KUKA KRL program: EPS_2_251112_SAMH01_A_20250918124112.src

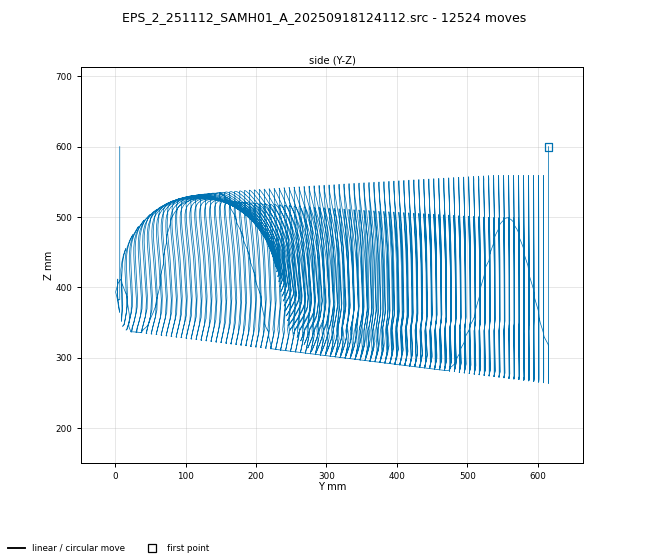
[picture p0: tool path of EPS_2_251112_SAMH01_A_20250918124112.src, 12524 of 12526 moves have a stored position in this frame; points joined in program order, loops and branches not executed]
&ACCESS RVP
&REL 4
&COMMENT QRS 19112012
&PARAM EDITMASK = *
DEF PART()
EXT BAS (BAS_COMMAND :IN,REAL :IN )
INT I
BAS (#INITMOV,0 )

;KUKA QRS Post kuka4.cps  Date:22-06-2017 !

File_ID=2848

QRS_PRE_INIT()

;Init var - Until changes are made in qrs_pre_init
Outlet_Square_prg=0
Inlet_1_Square_prg=0
Inlet_2_Square_prg=0
Inlet_3_Square_prg=0
Inlet_4_Square_prg=0
Inlet_5_Square_prg=0

Outlet_1={X 0.000, Y 535.490, Z 458.500, B 0.000, E1 0.000 }
Inlet_1={X 0.000, Y 540.090, Z 424.000, B 0.000, E1 110.000 }
Outlet_1_type=201
Inlet_1_type=150
;QRS#1=Sidecore dimensions
;QRS#2=200-8" PVC SDR 35
;QRS#3=150-6" PVC SDR 28
;QRS#4=
;QRS#5=
;QRS#6=
;QRS#7=
;QRS#8=
;QRS#9=12-08 PSX
;QRS#10=10-06 PSX
;QRS#11=
;QRS#12=
;QRS#13=
;QRS#14=
;QRS#15=
;QRS#16=1220x127x838 2,75'
;QRS#17=EPS Height
;QRS#18=559
;QRS#19=*
;QRS#20= UPDATED VERSION 22-06-2017
;QRS#21=*
Outlet_Square=0100
Inlet_1_Square=070
Inlet_2_Square=0
Inlet_3_Square=0
Inlet_4_Square=0
Inlet_5_Square=0
Mill_Square=1
Outlet_Square_Prg=204
Inlet_1_Square_prg=203

QRS_INIT()

$ADVANCE=5

; T1
PTP {E1 173.706,E2 173.706}
PTP {X 0,Y 615.438,A -85,B 0,C 180,E1 173.706,E2 173.706,E3 0,E4 0,E5 0,E6 0}
QRS_SPEED_INIT()
LIN {X 0,Y 615.438,Z 600,A -85,B 0,C 180,E1 173.706,E2 173.706,E3 0,E4 0,E5 0,E6 0} C_VEL
LIN {X 0,Y 615.438,Z 326.206,A -85,B 0,C 180,E1 173.706,E2 173.706} C_VEL
LIN {X 0,Y 615.438,Z 317.812,A -85,B 0,C 180,E1 173.706,E2 173.706} C_VEL
LIN {X 0,Y 615.44,Z 316.11,A -85,B 0,C 180,E1 173.422,E2 173.422} C_VEL
LIN {X 0,Y 615.492,Z 334.71,A -85,B 0,C 180,E1 170.635,E2 170.635} C_VEL
LIN {X 0,Y 615.479,Z 338.467,A -85,B 0,C 180,E1 170.075,E2 170.075} C_VEL
LIN {X 0,Y 615.469,Z 414.985,A -85,B 0,C 180,E1 169.169,E2 169.169} C_VEL
LIN {X 0,Y 615.464,Z 424.01,A -85,B 0,C 180,E1 168.989,E2 168.989} C_VEL
LIN {X 0,Y 615.468,Z 433.065,A -85,B 0,C 180,E1 168.723,E2 168.723} C_VEL
LIN {X 0,Y 615.491,Z 441.502,A -85,B 0,C 180,E1 168.389,E2 168.389} C_VEL
LIN {X 0,Y 615.495,Z 449.816,A -85,B 0,C 180,E1 167.972,E2 167.972} C_VEL
LIN {X 0,Y 615.478,Z 457.873,A -85,B 0,C 180,E1 167.469,E2 167.469} C_VEL
LIN {X 0,Y 615.498,Z 466.559,A -85,B 0,C 180,E1 166.799,E2 166.799} C_VEL
LIN {X 0,Y 615.497,Z 474.267,A -85,B 0,C 180,E1 166.046,E2 166.046} C_VEL
LIN {X 0,Y 615.495,Z 480.527,A -85,B 0,C 180,E1 165.282,E2 165.282} C_VEL
LIN {X 0,Y 615.495,Z 484.105,A -85,B 0,C 180,E1 164.774,E2 164.774} C_VEL
LIN {X 0,Y 615.494,Z 489.374,A -85,B 0,C 180,E1 163.824,E2 163.824} C_VEL
LIN {X 0,Y 615.496,Z 492.626,A -85,B 0,C 180,E1 163.072,E2 163.072} C_VEL
LIN {X 0,Y 615.496,Z 495.783,A -85,B 0,C 180,E1 162.043,E2 162.043} C_VEL
LIN {X 0,Y 615.487,Z 497.204,A -85,B 0,C 180,E1 161.354,E2 161.354} C_VEL
LIN {X 0,Y 615.491,Z 498.08,A -85,B 0,C 180,E1 160.662,E2 160.662} C_VEL
LIN {X 0,Y 615.494,Z 498.389,A -85,B 0,C 180,E1 159.967,E2 159.967} C_VEL
LIN {X 0,Y 615.492,Z 498.089,A -85,B 0,C 180,E1 159.269,E2 159.269} C_VEL
LIN {X 0,Y 615.493,Z 497.219,A -85,B 0,C 180,E1 158.568,E2 158.568} C_VEL
LIN {X 0,Y 615.496,Z 495.238,A -85,B 0,C 180,E1 157.642,E2 157.642} C_VEL
LIN {X 0,Y 615.491,Z 492.494,A -85,B 0,C 180,E1 156.8,E2 156.8} C_VEL
LIN {X 0,Y 615.495,Z 487.553,A -85,B 0,C 180,E1 155.728,E2 155.728} C_VEL
LIN {X 0,Y 615.494,Z 482.185,A -85,B 0,C 180,E1 154.861,E2 154.861} C_VEL
LIN {X 0,Y 615.494,Z 476.317,A -85,B 0,C 180,E1 154.102,E2 154.102} C_VEL
LIN {X 0,Y 615.495,Z 469.696,A -85,B 0,C 180,E1 153.403,E2 153.403} C_VEL
LIN {X 0,Y 615.481,Z 460.735,A -85,B 0,C 180,E1 152.638,E2 152.638} C_VEL
LIN {X 0,Y 615.489,Z 451.227,A -85,B 0,C 180,E1 152.017,E2 152.017} C_VEL
LIN {X 0,Y 615.493,Z 443.482,A -85,B 0,C 180,E1 151.609,E2 151.609} C_VEL
LIN {X 0,Y 615.485,Z 434.82,A -85,B 0,C 180,E1 151.248,E2 151.248} C_VEL
LIN {X 0,Y 615.475,Z 425.873,A -85,B 0,C 180,E1 150.967,E2 150.967} C_VEL
LIN {X 0,Y 615.475,Z 417.455,A -85,B 0,C 180,E1 150.78,E2 150.78} C_VEL
LIN {X 0,Y 615.484,Z 393.949,A -85,B 0,C 180,E1 150.482,E2 150.482} C_VEL
LIN {X 0,Y 615.474,Z 338.415,A -85,B 0,C 180,E1 149.827,E2 149.827} C_VEL
LIN {X 0,Y 615.477,Z 319.226,A -85,B 0,C 180,E1 146.958,E2 146.958} C_VEL
LIN {X 0,Y 615.479,Z 300.718,A -85,B 0,C 180,E1 144.162,E2 144.162} C_VEL
LIN {X 0,Y 615.449,Z 283.396,A -85,B 0,C 180,E1 141.511,E2 141.511} C_VEL
LIN {X 0,Y 615.497,Z 265.36,A -85,B 0,C 180,E1 138.714,E2 138.714} C_VEL
LIN {X 0,Y 615.465,Z 263.688,A -85,B 0,C 180,E1 138.449,E2 138.449} C_VEL
LIN {X 0,Y 615.43,Z 263.692,A -85,B 0,C 180,E1 135.845,E2 135.845} C_VEL
LIN {X 0,Y 615.44,Z 263.696,A -85,B 0,C 180,E1 133.245,E2 133.245} C_VEL
LIN {X 0,Y 615.487,Z 263.703,A -85,B 0,C 180,E1 130.603,E2 130.603} C_VEL
LIN {X 0,Y 615.477,Z 263.689,A -85,B 0,C 180,E1 128.01,E2 128.01} C_VEL
LIN {X 0,Y 615.451,Z 263.69,A -85,B 0,C 180,E1 125.616,E2 125.616} C_VEL
LIN {X 0,Y 615.432,Z 263.692,A -85,B 0,C 180,E1 123.237,E2 123.237} C_VEL
LIN {X 0,Y 615.427,Z 263.693,A -85,B 0,C 180,E1 120.921,E2 120.921} C_VEL
LIN {X 0,Y 615.427,Z 263.694,A -85,B 0,C 180,E1 118.659,E2 118.659} C_VEL
LIN {X 0,Y 615.499,Z 263.699,A -85,B 0,C 180,E1 115.714,E2 115.714} C_VEL
LIN {X 0,Y 615.444,Z 263.691,A -85,B 0,C 180,E1 112.845,E2 112.845} C_VEL
LIN {X 0,Y 615.431,Z 263.692,A -85,B 0,C 180,E1 110.542,E2 110.542} C_VEL
LIN {X 0,Y 615.442,Z 263.691,A -85,B 0,C 180,E1 108.591,E2 108.591} C_VEL
LIN {X 0,Y 615.437,Z 263.691,A -85,B 0,C 180,E1 106.414,E2 106.414} C_VEL
LIN {X 0,Y 615.461,Z 263.69,A -85,B 0,C 180,E1 104.55,E2 104.55} C_VEL
LIN {X 0,Y 615.424,Z 263.694,A -85,B 0,C 180,E1 101.862,E2 101.862} C_VEL
LIN {X 0,Y 615.426,Z 263.693,A -85,B 0,C 180,E1 99.864,E2 99.864} C_VEL
LIN {X 0,Y 615.432,Z 263.692,A -85,B 0,C 180,E1 97.877,E2 97.877} C_VEL
LIN {X 0,Y 615.442,Z 263.691,A -85,B 0,C 180,E1 95.9,E2 95.9} C_VEL
LIN {X 0,Y 615.457,Z 263.691,A -85,B 0,C 180,E1 93.93,E2 93.93} C_VEL
LIN {X 0,Y 615.423,Z 263.694,A -85,B 0,C 180,E1 91.31,E2 91.31} C_VEL
LIN {X 0,Y 615.428,Z 263.693,A -85,B 0,C 180,E1 89.347,E2 89.347} C_VEL
LIN {X 0,Y 615.438,Z 263.692,A -85,B 0,C 180,E1 87.384,E2 87.384} C_VEL
LIN {X 0,Y 615.452,Z 263.691,A -85,B 0,C 180,E1 85.417,E2 85.417} C_VEL
LIN {X 0,Y 615.421,Z 263.694,A -85,B 0,C 180,E1 82.786,E2 82.786} C_VEL
LIN {X 0,Y 615.424,Z 263.694,A -85,B 0,C 180,E1 80.803,E2 80.803} C_VEL
LIN {X 0,Y 615.43,Z 263.693,A -85,B 0,C 180,E1 78.808,E2 78.808} C_VEL
LIN {X 0,Y 615.437,Z 263.693,A -85,B 0,C 180,E1 76.8,E2 76.8} C_VEL
LIN {X 0,Y 615.446,Z 263.692,A -85,B 0,C 180,E1 74.776,E2 74.776} C_VEL
LIN {X 0,Y 615.453,Z 263.692,A -85,B 0,C 180,E1 72.732,E2 72.732} C_VEL
LIN {X 0,Y 615.459,Z 263.692,A -85,B 0,C 180,E1 70.665,E2 70.665} C_VEL
LIN {X 0,Y 615.462,Z 263.692,A -85,B 0,C 180,E1 68.571,E2 68.571} C_VEL
LIN {X 0,Y 615.423,Z 263.694,A -85,B 0,C 180,E1 66.006,E2 66.006} C_VEL
LIN {X 0,Y 615.418,Z 263.696,A -85,B 0,C 180,E1 63.557,E2 63.557} C_VEL
LIN {X 0,Y 615.49,Z 263.702,A -85,B 0,C 180,E1 60.599,E2 60.599} C_VEL
LIN {X 0,Y 615.431,Z 263.694,A -85,B 0,C 180,E1 57.678,E2 57.678} C_VEL
LIN {X 0,Y 615.416,Z 263.696,A -85,B 0,C 180,E1 55.186,E2 55.186} C_VEL
LIN {X 0,Y 615.416,Z 263.696,A -85,B 0,C 180,E1 53.073,E2 53.073} C_VEL
LIN {X 0,Y 615.415,Z 263.696,A -85,B 0,C 180,E1 50.947,E2 50.947} C_VEL
LIN {X 0,Y 615.416,Z 263.695,A -85,B 0,C 180,E1 48.914,E2 48.914} C_VEL
LIN {X 0,Y 615.414,Z 263.696,A -85,B 0,C 180,E1 46.756,E2 46.756} C_VEL
LIN {X 0,Y 615.427,Z 263.694,A -85,B 0,C 180,E1 44.933,E2 44.933} C_VEL
LIN {X 0,Y 615.415,Z 263.696,A -85,B 0,C 180,E1 42.36,E2 42.36} C_VEL
LIN {X 0,Y 615.417,Z 263.698,A -85,B 0,C 180,E1 40.09,E2 40.09} C_VEL
LIN {X 0,Y 615.417,Z 263.697,A -85,B 0,C 180,E1 38.013,E2 38.013} C_VEL
LIN {X 0,Y 615.433,Z 263.698,A -85,B 0,C 180,E1 35.62,E2 35.62} C_VEL
LIN {X 0,Y 615.46,Z 263.7,A -85,B 0,C 180,E1 33.238,E2 33.238} C_VEL
LIN {X 0,Y 615.488,Z 263.701,A -85,B 0,C 180,E1 30.92,E2 30.92} C_VEL
LIN {X 0,Y 615.475,Z 263.694,A -85,B 0,C 180,E1 28.462,E2 28.462} C_VEL
LIN {X 0,Y 615.416,Z 263.696,A -85,B 0,C 180,E1 25.719,E2 25.719} C_VEL
LIN {X 0,Y 615.414,Z 263.696,A -85,B 0,C 180,E1 23.56,E2 23.56} C_VEL
LIN {X 0,Y 615.413,Z 263.696,A -85,B 0,C 180,E1 21.435,E2 21.435} C_VEL
LIN {X 0,Y 615.411,Z 263.697,A -85,B 0,C 180,E1 19.341,E2 19.341} C_VEL
LIN {X 0,Y 615.416,Z 263.696,A -85,B 0,C 180,E1 17.273,E2 17.273} C_VEL
LIN {X 0,Y 615.42,Z 263.696,A -85,B 0,C 180,E1 15.228,E2 15.228} C_VEL
LIN {X 0,Y 615.426,Z 263.696,A -85,B 0,C 180,E1 13.203,E2 13.203} C_VEL
LIN {X 0,Y 615.414,Z 263.697,A -85,B 0,C 180,E1 10.889,E2 10.889} C_VEL
LIN {X 0,Y 615.407,Z 263.697,A -85,B 0,C 180,E1 8.538,E2 8.538} C_VEL
LIN {X 0,Y 615.41,Z 263.697,A -85,B 0,C 180,E1 6.558,E2 6.558} C_VEL
LIN {X 0,Y 615.415,Z 263.697,A -85,B 0,C 180,E1 4.585,E2 4.585} C_VEL
LIN {X 0,Y 615.425,Z 263.696,A -85,B 0,C 180,E1 2.618,E2 2.618} C_VEL
LIN {X 0,Y 615.44,Z 263.696,A -85,B 0,C 180,E1 0.655,E2 0.655} C_VEL
LIN {X 0,Y 615.406,Z 263.698,A -85,B 0,C 180,E1 -1.963,E2 -1.963} C_VEL
LIN {X 0,Y 615.41,Z 263.698,A -85,B 0,C 180,E1 -3.929,E2 -3.929} C_VEL
LIN {X 0,Y 615.419,Z 263.697,A -85,B 0,C 180,E1 -5.899,E2 -5.899} C_VEL
LIN {X 0,Y 615.431,Z 263.697,A -85,B 0,C 180,E1 -7.876,E2 -7.876} C_VEL
LIN {X 0,Y 615.448,Z 263.697,A -85,B 0,C 180,E1 -9.862,E2 -9.862} C_VEL
LIN {X 0,Y 615.406,Z 263.698,A -85,B 0,C 180,E1 -12.531,E2 -12.531} C_VEL
LIN {X 0,Y 615.409,Z 263.698,A -85,B 0,C 180,E1 -14.551,E2 -14.551} C_VEL
LIN {X 0,Y 615.412,Z 263.698,A -85,B 0,C 180,E1 -16.588,E2 -16.588} C_VEL
LIN {X 0,Y 615.416,Z 263.698,A -85,B 0,C 180,E1 -18.648,E2 -18.648} C_VEL
LIN {X 0,Y 615.418,Z 263.698,A -85,B 0,C 180,E1 -20.733,E2 -20.733} C_VEL
LIN {X 0,Y 615.418,Z 263.698,A -85,B 0,C 180,E1 -22.847,E2 -22.847} C_VEL
LIN {X 0,Y 615.416,Z 263.698,A -85,B 0,C 180,E1 -24.994,E2 -24.994} C_VEL
LIN {X 0,Y 615.411,Z 263.698,A -85,B 0,C 180,E1 -27.18,E2 -27.18} C_VEL
LIN {X 0,Y 615.405,Z 263.698,A -85,B 0,C 180,E1 -29.41,E2 -29.41} C_VEL
LIN {X 0,Y 615.399,Z 263.699,A -85,B 0,C 180,E1 -31.69,E2 -31.69} C_VEL
LIN {X 0,Y 615.403,Z 263.699,A -85,B 0,C 180,E1 -34.027,E2 -34.027} C_VEL
LIN {X 0,Y 615.416,Z 263.7,A -85,B 0,C 180,E1 -36.429,E2 -36.429} C_VEL
LIN {X 0,Y 615.489,Z 263.7,A -85,B 0,C 180,E1 -39.071,E2 -39.071} C_VEL
LIN {X 0,Y 615.469,Z 263.699,A -85,B 0,C 180,E1 -41.475,E2 -41.475} C_VEL
LIN {X 0,Y 615.407,Z 263.699,A -85,B 0,C 180,E1 -44.156,E2 -44.156} C_VEL
LIN {X 0,Y 615.401,Z 263.699,A -85,B 0,C 180,E1 -46.755,E2 -46.755} C_VEL
LIN {X 0,Y 615.401,Z 263.699,A -85,B 0,C 180,E1 -48.526,E2 -48.526} C_VEL
LIN {X 0,Y 615.427,Z 263.699,A -85,B 0,C 180,E1 -50.252,E2 -50.252} C_VEL
LIN {X 0,Y 615.476,Z 263.7,A -85,B 0,C 180,E1 -51.989,E2 -51.989} C_VEL
LIN {X 0,Y 615.439,Z 263.7,A -85,B 0,C 180,E1 -54.387,E2 -54.387} C_VEL
LIN {X 0,Y 615.412,Z 263.7,A -85,B 0,C 180,E1 -56.765,E2 -56.765} C_VEL
LIN {X 0,Y 615.4,Z 263.7,A -85,B 0,C 180,E1 -59.08,E2 -59.08} C_VEL
LIN {X 0,Y 615.396,Z 263.7,A -85,B 0,C 180,E1 -61.342,E2 -61.342} C_VEL
LIN {X 0,Y 615.396,Z 263.7,A -85,B 0,C 180,E1 -63.556,E2 -63.556} C_VEL
LIN {X 0,Y 615.397,Z 263.7,A -85,B 0,C 180,E1 -65.728,E2 -65.728} C_VEL
LIN {X 0,Y 615.404,Z 263.876,A -85,B 0,C 180,E1 -68.041,E2 -68.041} C_VEL
LIN {X 0,Y 615.485,Z 285.488,A -85,B 0,C 180,E1 -70.492,E2 -70.492} C_VEL
LIN {X 0,Y 615.477,Z 311.706,A -85,B 0,C 180,E1 -73.416,E2 -73.416} C_VEL
LIN {X 0,Y 615.462,Z 336.351,A -85,B 0,C 180,E1 -76.128,E2 -76.128} C_VEL
LIN {X 0,Y 615.487,Z 345.547,A -85,B 0,C 180,E1 -77.116,E2 -77.116} C_VEL
LIN {X 0,Y 615.464,Z 454.974,A -85,B 0,C 180,E1 -78.413,E2 -78.413} C_VEL
LIN {X 0,Y 615.461,Z 467.439,A -85,B 0,C 180,E1 -78.684,E2 -78.684} C_VEL
LIN {X 0,Y 615.484,Z 480.6,A -85,B 0,C 180,E1 -79.112,E2 -79.112} C_VEL
LIN {X 0,Y 615.48,Z 492.524,A -85,B 0,C 180,E1 -79.642,E2 -79.642} C_VEL
LIN {X 0,Y 615.473,Z 502.758,A -85,B 0,C 180,E1 -80.223,E2 -80.223} C_VEL
LIN {X 0,Y 615.498,Z 513.248,A -85,B 0,C 180,E1 -80.969,E2 -80.969} C_VEL
LIN {X 0,Y 615.498,Z 521.025,A -85,B 0,C 180,E1 -81.631,E2 -81.631} C_VEL
LIN {X 0,Y 615.494,Z 529.082,A -85,B 0,C 180,E1 -82.457,E2 -82.457} C_VEL
LIN {X 0,Y 615.494,Z 537.084,A -85,B 0,C 180,E1 -83.445,E2 -83.445} C_VEL
LIN {X 0,Y 615.499,Z 543.415,A -85,B 0,C 180,E1 -84.432,E2 -84.432} C_VEL
LIN {X 0,Y 615.498,Z 548.449,A -85,B 0,C 180,E1 -85.417,E2 -85.417} C_VEL
LIN {X 0,Y 615.496,Z 552.355,A -85,B 0,C 180,E1 -86.401,E2 -86.401} C_VEL
LIN {X 0,Y 615.497,Z 555.237,A -85,B 0,C 180,E1 -87.384,E2 -87.384} C_VEL
LIN {X 0,Y 615.496,Z 556.611,A -85,B 0,C 180,E1 -88.038,E2 -88.038} C_VEL
LIN {X 0,Y 615.495,Z 557.582,A -85,B 0,C 180,E1 -88.693,E2 -88.693} C_VEL
LIN {X 0,Y 615.488,Z 558.39,A -85,B 0,C 180,E1 -90.001,E2 -90.001} C_VEL
LIN {X 0,Y 615.495,Z 557.579,A -85,B 0,C 180,E1 -91.31,E2 -91.31} C_VEL
LIN {X 0,Y 615.496,Z 556.606,A -85,B 0,C 180,E1 -91.964,E2 -91.964} C_VEL
LIN {X 0,Y 615.497,Z 555.23,A -85,B 0,C 180,E1 -92.619,E2 -92.619} C_VEL
LIN {X 0,Y 615.496,Z 552.346,A -85,B 0,C 180,E1 -93.602,E2 -93.602} C_VEL
LIN {X 0,Y 615.498,Z 548.438,A -85,B 0,C 180,E1 -94.585,E2 -94.585} C_VEL
LIN {X 0,Y 615.499,Z 543.401,A -85,B 0,C 180,E1 -95.57,E2 -95.57} C_VEL
LIN {X 0,Y 615.494,Z 536.852,A -85,B 0,C 180,E1 -96.586,E2 -96.586} C_VEL
LIN {X 0,Y 615.493,Z 529.059,A -85,B 0,C 180,E1 -97.546,E2 -97.546} C_VEL
LIN {X 0,Y 615.498,Z 520.997,A -85,B 0,C 180,E1 -98.372,E2 -98.372} C_VEL
LIN {X 0,Y 615.498,Z 509.991,A -85,B 0,C 180,E1 -99.282,E2 -99.282} C_VEL
LIN {X 0,Y 615.468,Z 498.573,A -85,B 0,C 180,E1 -100.029,E2 -100.029} C_VEL
LIN {X 0,Y 615.49,Z 487.115,A -85,B 0,C 180,E1 -100.617,E2 -100.617} C_VEL
LIN {X 0,Y 615.469,Z 475.315,A -85,B 0,C 180,E1 -101.079,E2 -101.079} C_VEL
LIN {X 0,Y 615.461,Z 462.237,A -85,B 0,C 180,E1 -101.444,E2 -101.444} C_VEL
LIN {X 0,Y 615.468,Z 448.932,A -85,B 0,C 180,E1 -101.673,E2 -101.673} C_VEL
LIN {X 0,Y 615.487,Z 345.364,A -85,B 0,C 180,E1 -102.886,E2 -102.886} C_VEL
LIN {X 0,Y 615.481,Z 319.385,A -85,B 0,C 180,E1 -105.735,E2 -105.735} C_VEL
LIN {X 0,Y 615.488,Z 294.967,A -85,B 0,C 180,E1 -108.445,E2 -108.445} C_VEL
LIN {X 0,Y 615.491,Z 271.57,A -85,B 0,C 180,E1 -111.08,E2 -111.08} C_VEL
LIN {X 0,Y 615.406,Z 263.7,A -85,B 0,C 180,E1 -112.006,E2 -112.006} C_VEL
LIN {X 0,Y 615.408,Z 263.698,A -85,B 0,C 180,E1 -114.274,E2 -114.274} C_VEL
LIN {X 0,Y 615.414,Z 263.698,A -85,B 0,C 180,E1 -116.446,E2 -116.446} C_VEL
LIN {X 0,Y 615.491,Z 263.702,A -85,B 0,C 180,E1 -119.404,E2 -119.404} C_VEL
LIN {X 0,Y 615.438,Z 263.692,A -85,B 0,C 180,E1 -122.324,E2 -122.324} C_VEL
LIN {X 0,Y 615.433,Z 263.693,A -85,B 0,C 180,E1 -124.694,E2 -124.694} C_VEL
LIN {X 0,Y 615.437,Z 263.694,A -85,B 0,C 180,E1 -126.931,E2 -126.931} C_VEL
LIN {X 0,Y 615.441,Z 263.694,A -85,B 0,C 180,E1 -129.057,E2 -129.057} C_VEL
LIN {X 0,Y 615.466,Z 263.697,A -85,B 0,C 180,E1 -131.472,E2 -131.472} C_VEL
LIN {X 0,Y 615.489,Z 263.691,A -85,B 0,C 180,E1 -134.146,E2 -134.146} C_VEL
LIN {X 0,Y 615.466,Z 263.685,A -85,B 0,C 180,E1 -136.951,E2 -136.951} C_VEL
LIN {X 0,Y 615.459,Z 263.691,A -85,B 0,C 180,E1 -139.392,E2 -139.392} C_VEL
LIN {X 0,Y 615.479,Z 263.701,A -85,B 0,C 180,E1 -141.984,E2 -141.984} C_VEL
LIN {X 0,Y 615.484,Z 263.694,A -85,B 0,C 180,E1 -144.384,E2 -144.384} C_VEL
LIN {X 0,Y 615.478,Z 263.687,A -85,B 0,C 180,E1 -146.764,E2 -146.764} C_VEL
LIN {X 0,Y 615.481,Z 263.683,A -85,B 0,C 180,E1 -149.08,E2 -149.08} C_VEL
LIN {X 0,Y 615.487,Z 263.681,A -85,B 0,C 180,E1 -151.542,E2 -151.542} C_VEL
LIN {X 0,Y 615.499,Z 263.7,A -85,B 0,C 180,E1 -154.42,E2 -154.42} C_VEL
LIN {X 0,Y 615.463,Z 263.689,A -85,B 0,C 180,E1 -157.155,E2 -157.155} C_VEL
LIN {X 0,Y 615.463,Z 263.686,A -85,B 0,C 180,E1 -159.438,E2 -159.438} C_VEL
LIN {X 0,Y 615.492,Z 263.683,A -85,B 0,C 180,E1 -162.044,E2 -162.044} C_VEL
LIN {X 0,Y 615.488,Z 263.702,A -85,B 0,C 180,E1 -164.774,E2 -164.774} C_VEL
LIN {X 0,Y 615.446,Z 263.693,A -85,B 0,C 180,E1 -167.469,E2 -167.469} C_VEL
LIN {X 0,Y 615.444,Z 263.694,A -85,B 0,C 180,E1 -169.473,E2 -169.473} C_VEL
LIN {X 0,Y 615.444,Z 263.696,A -85,B 0,C 180,E1 -171.463,E2 -171.463} C_VEL
LIN {X 0,Y 615.446,Z 263.697,A -85,B 0,C 180,E1 -173.443,E2 -173.443} C_VEL
LIN {X 0,Y 615.452,Z 263.698,A -85,B 0,C 180,E1 -175.416,E2 -175.416} C_VEL
LIN {X 0,Y 615.461,Z 263.699,A -85,B 0,C 180,E1 -177.382,E2 -177.382} C_VEL
LIN {X 0,Y 615.449,Z 263.876,A -85,B 0,C 180,E1 -178.569,E2 -178.569} C_VEL
LIN {X 0,Y 615.464,Z 282.556,A -85,B 0,C 180,E1 -181.473,E2 -181.473} C_VEL
LIN {X 0,Y 615.49,Z 299.668,A -85,B 0,C 180,E1 -184.093,E2 -184.093} C_VEL
LIN {X 0,Y 615.44,Z 316.11,A -85,B 0,C 180,E1 -186.578,E2 -186.578} C_VEL
LIN {X 0,Y 614.801,Z 319.34,A -85,B 0,C 180,E1 -187.038,E2 -187.038} C_VEL
LIN {X 0,Y 609.131,Z 330.029,A -85,B 0,C 180,E1 -188.511,E2 -188.511} C_VEL
LIN {X 0,Y 608.462,Z 333.199,A -85,B 0,C 180,E1 -188.977,E2 -188.977} C_VEL
LIN {X 0,Y 608.47,Z 338.969,A -85,B 0,C 180,E1 -189.809,E2 -189.809} C_VEL
LIN {X 0,Y 608.485,Z 416.005,A -85,B 0,C 180,E1 -190.732,E2 -190.732} C_VEL
LIN {X 0,Y 608.476,Z 425.448,A -85,B 0,C 180,E1 -190.933,E2 -190.933} C_VEL
LIN {X 0,Y 608.477,Z 435.819,A -85,B 0,C 180,E1 -191.26,E2 -191.26} C_VEL
LIN {X 0,Y 608.496,Z 446.774,A -85,B 0,C 180,E1 -191.746,E2 -191.746} C_VEL
LIN {X 0,Y 608.446,Z 456.699,A -85,B 0,C 180,E1 -192.339,E2 -192.339} C_VEL
LIN {X 0,Y 608.474,Z 464.636,A -85,B 0,C 180,E1 -192.932,E2 -192.932} C_VEL
LIN {X 0,Y 608.458,Z 471.217,A -85,B 0,C 180,E1 -193.527,E2 -193.527} C_VEL
LIN {X 0,Y 608.447,Z 477.478,A -85,B 0,C 180,E1 -194.209,E2 -194.209} C_VEL
LIN {X 0,Y 608.436,Z 483.883,A -85,B 0,C 180,E1 -195.064,E2 -195.064} C_VEL
LIN {X 0,Y 608.454,Z 489.737,A -85,B 0,C 180,E1 -196.094,E2 -196.094} C_VEL
LIN {X 0,Y 608.445,Z 492.812,A -85,B 0,C 180,E1 -196.785,E2 -196.785} C_VEL
LIN {X 0,Y 608.434,Z 495.206,A -85,B 0,C 180,E1 -197.477,E2 -197.477} C_VEL
LIN {X 0,Y 608.433,Z 496.953,A -85,B 0,C 180,E1 -198.173,E2 -198.173} C_VEL
LIN {X 0,Y 608.421,Z 498.146,A -85,B 0,C 180,E1 -198.871,E2 -198.871} C_VEL
LIN {X 0,Y 608.409,Z 498.802,A -85,B 0,C 180,E1 -199.572,E2 -199.572} C_VEL
LIN {X 0,Y 608.43,Z 498.726,A -85,B 0,C 180,E1 -200.681,E2 -200.681} C_VEL
LIN {X 0,Y 608.424,Z 497.455,A -85,B 0,C 180,E1 -201.694,E2 -201.694} C_VEL
LIN {X 0,Y 608.435,Z 494.677,A -85,B 0,C 180,E1 -202.767,E2 -202.767} C_VEL
LIN {X 0,Y 608.445,Z 492.072,A -85,B 0,C 180,E1 -203.485,E2 -203.485} C_VEL
LIN {X 0,Y 608.437,Z 488.03,A -85,B 0,C 180,E1 -204.328,E2 -204.328} C_VEL
LIN {X 0,Y 608.453,Z 483.226,A -85,B 0,C 180,E1 -205.118,E2 -205.118} C_VEL
LIN {X 0,Y 608.453,Z 477.934,A -85,B 0,C 180,E1 -205.828,E2 -205.828} C_VEL
LIN {X 0,Y 608.468,Z 470.954,A -85,B 0,C 180,E1 -206.589,E2 -206.589} C_VEL
LIN {X 0,Y 608.465,Z 463.97,A -85,B 0,C 180,E1 -207.213,E2 -207.213} C_VEL
LIN {X 0,Y 608.453,Z 454.639,A -85,B 0,C 180,E1 -207.892,E2 -207.892} C_VEL
LIN {X 0,Y 608.486,Z 443.683,A -85,B 0,C 180,E1 -208.493,E2 -208.493} C_VEL
LIN {X 0,Y 608.477,Z 434.015,A -85,B 0,C 180,E1 -208.893,E2 -208.893} C_VEL
LIN {X 0,Y 608.49,Z 424.806,A -85,B 0,C 180,E1 -209.173,E2 -209.173} C_VEL
LIN {X 0,Y 608.48,Z 416.403,A -85,B 0,C 180,E1 -209.351,E2 -209.351} C_VEL
LIN {X 0,Y 608.451,Z 338.704,A -85,B 0,C 180,E1 -210.288,E2 -210.288} C_VEL
LIN {X 0,Y 608.453,Z 318.865,A -85,B 0,C 180,E1 -213.275,E2 -213.275} C_VEL
LIN {X 0,Y 608.478,Z 300.385,A -85,B 0,C 180,E1 -216.091,E2 -216.091} C_VEL
LIN {X 0,Y 608.476,Z 284.212,A -85,B 0,C 180,E1 -218.588,E2 -218.588} C_VEL
LIN {X 0,Y 608.53,Z 265.787,A -85,B 0,C 180,E1 -221.477,E2 -221.477} C_VEL
LIN {X 0,Y 608.439,Z 264.69,A -85,B 0,C 180,E1 -221.677,E2 -221.677} C_VEL
LIN {X 0,Y 608.432,Z 264.689,A -85,B 0,C 180,E1 -223.873,E2 -223.873} C_VEL
LIN {X 0,Y 608.431,Z 264.691,A -85,B 0,C 180,E1 -226.696,E2 -226.696} C_VEL
LIN {X 0,Y 608.408,Z 264.694,A -85,B 0,C 180,E1 -228.823,E2 -228.823} C_VEL
LIN {X 0,Y 608.445,Z 264.697,A -85,B 0,C 180,E1 -231.413,E2 -231.413} C_VEL
LIN {X 0,Y 608.469,Z 264.69,A -85,B 0,C 180,E1 -233.952,E2 -233.952} C_VEL
LIN {X 0,Y 608.435,Z 264.691,A -85,B 0,C 180,E1 -236.33,E2 -236.33} C_VEL
LIN {X 0,Y 608.426,Z 264.689,A -85,B 0,C 180,E1 -238.736,E2 -238.736} C_VEL
LIN {X 0,Y 608.404,Z 264.692,A -85,B 0,C 180,E1 -240.978,E2 -240.978} C_VEL
LIN {X 0,Y 608.397,Z 264.692,A -85,B 0,C 180,E1 -243.225,E2 -243.225} C_VEL
LIN {X 0,Y 608.413,Z 264.691,A -85,B 0,C 180,E1 -245.428,E2 -245.428} C_VEL
LIN {X 0,Y 608.456,Z 264.694,A -85,B 0,C 180,E1 -248.309,E2 -248.309} C_VEL
LIN {X 0,Y 608.425,Z 264.691,A -85,B 0,C 180,E1 -251.298,E2 -251.298} C_VEL
LIN {X 0,Y 608.409,Z 264.691,A -85,B 0,C 180,E1 -253.905,E2 -253.905} C_VEL
LIN {X 0,Y 608.438,Z 264.693,A -85,B 0,C 180,E1 -256.643,E2 -256.643} C_VEL
LIN {X 0,Y 608.463,Z 264.692,A -85,B 0,C 180,E1 -259.35,E2 -259.35} C_VEL
LIN {X 0,Y 608.407,Z 264.692,A -85,B 0,C 180,E1 -262.032,E2 -262.032} C_VEL
LIN {X 0,Y 608.424,Z 264.691,A -85,B 0,C 180,E1 -264.032,E2 -264.032} C_VEL
LIN {X 0,Y 608.428,Z 264.691,A -85,B 0,C 180,E1 -266.025,E2 -266.025} C_VEL
LIN {X 0,Y 608.446,Z 264.691,A -85,B 0,C 180,E1 -268.013,E2 -268.013} C_VEL
LIN {X 0,Y 608.407,Z 264.691,A -85,B 0,C 180,E1 -270.66,E2 -270.66} C_VEL
LIN {X 0,Y 608.433,Z 264.689,A -85,B 0,C 180,E1 -272.647,E2 -272.647} C_VEL
LIN {X 0,Y 608.409,Z 264.692,A -85,B 0,C 180,E1 -275.3,E2 -275.3} C_VEL
LIN {X 0,Y 608.424,Z 264.697,A -85,B 0,C 180,E1 -277.965,E2 -277.965} C_VEL
LIN {X 0,Y 608.423,Z 264.692,A -85,B 0,C 180,E1 -280.931,E2 -280.931} C_VEL
LIN {X 0,Y 608.415,Z 264.69,A -85,B 0,C 180,E1 -283.355,E2 -283.355} C_VEL
LIN {X 0,Y 608.427,Z 264.689,A -85,B 0,C 180,E1 -285.404,E2 -285.404} C_VEL
LIN {X 0,Y 608.413,Z 264.691,A -85,B 0,C 180,E1 -287.475,E2 -287.475} C_VEL
LIN {X 0,Y 608.414,Z 264.691,A -85,B 0,C 180,E1 -289.568,E2 -289.568} C_VEL
LIN {X 0,Y 608.429,Z 264.689,A -85,B 0,C 180,E1 -291.689,E2 -291.689} C_VEL
LIN {X 0,Y 608.398,Z 264.692,A -85,B 0,C 180,E1 -294.135,E2 -294.135} C_VEL
LIN {X 0,Y 608.402,Z 264.692,A -85,B 0,C 180,E1 -296.033,E2 -296.033} C_VEL
LIN {X 0,Y 608.393,Z 264.693,A -85,B 0,C 180,E1 -298.265,E2 -298.265} C_VEL
LIN {X 0,Y 608.399,Z 264.692,A -85,B 0,C 180,E1 -300.544,E2 -300.544} C_VEL
LIN {X 0,Y 608.41,Z 264.692,A -85,B 0,C 180,E1 -302.877,E2 -302.877} C_VEL
LIN {X 0,Y 608.408,Z 264.695,A -85,B 0,C 180,E1 -305.274,E2 -305.274} C_VEL
LIN {X 0,Y 608.456,Z 264.691,A -85,B 0,C 180,E1 -308.238,E2 -308.238} C_VEL
LIN {X 0,Y 608.452,Z 264.692,A -85,B 0,C 180,E1 -310.328,E2 -310.328} C_VEL
LIN {X 0,Y 608.396,Z 264.693,A -85,B 0,C 180,E1 -312.958,E2 -312.958} C_VEL
LIN {X 0,Y 608.398,Z 264.693,A -85,B 0,C 180,E1 -315.198,E2 -315.198} C_VEL
LIN {X 0,Y 608.41,Z 264.693,A -85,B 0,C 180,E1 -317.036,E2 -317.036} C_VEL
LIN {X 0,Y 608.441,Z 264.693,A -85,B 0,C 180,E1 -318.822,E2 -318.822} C_VEL
LIN {X 0,Y 608.398,Z 264.693,A -85,B 0,C 180,E1 -321.406,E2 -321.406} C_VEL
LIN {X 0,Y 608.448,Z 264.692,A -85,B 0,C 180,E1 -323.084,E2 -323.084} C_VEL
LIN {X 0,Y 608.43,Z 264.69,A -85,B 0,C 180,E1 -325.528,E2 -325.528} C_VEL
LIN {X 0,Y 608.407,Z 264.691,A -85,B 0,C 180,E1 -327.902,E2 -327.902} C_VEL
LIN {X 0,Y 608.398,Z 264.692,A -85,B 0,C 180,E1 -330.216,E2 -330.216} C_VEL
LIN {X 0,Y 608.389,Z 264.694,A -85,B 0,C 180,E1 -332.479,E2 -332.479} C_VEL
LIN {X 0,Y 608.386,Z 264.695,A -85,B 0,C 180,E1 -334.696,E2 -334.696} C_VEL
LIN {X 0,Y 608.392,Z 264.694,A -85,B 0,C 180,E1 -336.873,E2 -336.873} C_VEL
LIN {X 0,Y 608.424,Z 264.694,A -85,B 0,C 180,E1 -339.313,E2 -339.313} C_VEL
LIN {X 0,Y 608.432,Z 264.7,A -85,B 0,C 180,E1 -341.827,E2 -341.827} C_VEL
LIN {X 0,Y 608.421,Z 264.692,A -85,B 0,C 180,E1 -344.592,E2 -344.592} C_VEL
LIN {X 0,Y 608.419,Z 264.693,A -85,B 0,C 180,E1 -346.642,E2 -346.642} C_VEL
LIN {X 0,Y 608.39,Z 264.693,A -85,B 0,C 180,E1 -349.348,E2 -349.348} C_VEL
LIN {X 0,Y 608.43,Z 264.693,A -85,B 0,C 180,E1 -352.032,E2 -352.032} C_VEL
LIN {X 0,Y 608.481,Z 264.692,A -85,B 0,C 180,E1 -354.698,E2 -354.698} C_VEL
LIN {X 0,Y 608.418,Z 264.692,A -85,B 0,C 180,E1 -357.351,E2 -357.351} C_VEL
LIN {X 0,Y 608.432,Z 264.692,A -85,B 0,C 180,E1 -359.338,E2 -359.338} C_VEL
LIN {X 0,Y 608.436,Z 264.693,A -85,B 0,C 180,E1 -361.323,E2 -361.323} C_VEL
LIN {X 0,Y 608.38,Z 264.695,A -85,B 0,C 180,E1 -363.974,E2 -363.974} C_VEL
LIN {X 0,Y 608.391,Z 264.694,A -85,B 0,C 180,E1 -365.967,E2 -365.967} C_VEL
LIN {X 0,Y 608.417,Z 264.692,A -85,B 0,C 180,E1 -367.967,E2 -367.967} C_VEL
LIN {X 0,Y 608.409,Z 264.694,A -85,B 0,C 180,E1 -369.978,E2 -369.978} C_VEL
LIN {X 0,Y 608.401,Z 264.692,A -85,B 0,C 180,E1 -372.678,E2 -372.678} C_VEL
LIN {X 0,Y 608.402,Z 264.692,A -85,B 0,C 180,E1 -374.722,E2 -374.722} C_VEL
LIN {X 0,Y 608.387,Z 264.694,A -85,B 0,C 180,E1 -376.786,E2 -376.786} C_VEL
LIN {X 0,Y 608.386,Z 264.694,A -85,B 0,C 180,E1 -378.871,E2 -378.871} C_VEL
LIN {X 0,Y 608.387,Z 264.694,A -85,B 0,C 180,E1 -380.984,E2 -380.984} C_VEL
LIN {X 0,Y 608.381,Z 264.695,A -85,B 0,C 180,E1 -383.126,E2 -383.126} C_VEL
LIN {X 0,Y 608.374,Z 264.695,A -85,B 0,C 180,E1 -385.304,E2 -385.304} C_VEL
LIN {X 0,Y 608.38,Z 264.695,A -85,B 0,C 180,E1 -387.521,E2 -387.521} C_VEL
LIN {X 0,Y 608.39,Z 264.694,A -85,B 0,C 180,E1 -389.783,E2 -389.783} C_VEL
LIN {X 0,Y 608.421,Z 264.697,A -85,B 0,C 180,E1 -392.528,E2 -392.528} C_VEL
LIN {X 0,Y 608.398,Z 264.698,A -85,B 0,C 180,E1 -395.28,E2 -395.28} C_VEL
LIN {X 0,Y 608.406,Z 264.692,A -85,B 0,C 180,E1 -397.75,E2 -397.75} C_VEL
LIN {X 0,Y 608.433,Z 264.694,A -85,B 0,C 180,E1 -399.442,E2 -399.442} C_VEL
LIN {X 0,Y 608.387,Z 264.694,A -85,B 0,C 180,E1 -402.067,E2 -402.067} C_VEL
LIN {X 0,Y 608.382,Z 264.695,A -85,B 0,C 180,E1 -404.264,E2 -404.264} C_VEL
LIN {X 0,Y 608.395,Z 264.693,A -85,B 0,C 180,E1 -406.698,E2 -406.698} C_VEL
LIN {X 0,Y 608.381,Z 264.694,A -85,B 0,C 180,E1 -408.666,E2 -408.666} C_VEL
LIN {X 0,Y 608.376,Z 264.695,A -85,B 0,C 180,E1 -410.713,E2 -410.713} C_VEL
LIN {X 0,Y 608.396,Z 264.693,A -85,B 0,C 180,E1 -412.85,E2 -412.85} C_VEL
LIN {X 0,Y 608.368,Z 264.696,A -85,B 0,C 180,E1 -415.105,E2 -415.105} C_VEL
LIN {X 0,Y 608.392,Z 264.694,A -85,B 0,C 180,E1 -417.487,E2 -417.487} C_VEL
LIN {X 0,Y 608.455,Z 264.695,A -85,B 0,C 180,E1 -420.225,E2 -420.225} C_VEL
LIN {X 0,Y 608.376,Z 264.696,A -85,B 0,C 180,E1 -423.227,E2 -423.227} C_VEL
LIN {X 0,Y 608.389,Z 264.694,A -85,B 0,C 180,E1 -425.43,E2 -425.43} C_VEL
LIN {X 0,Y 608.391,Z 264.841,A -85,B 0,C 180,E1 -427.886,E2 -427.886} C_VEL
LIN {X 0,Y 608.569,Z 279.706,A -85,B 0,C 180,E1 -429.602,E2 -429.602} C_VEL
LIN {X 0,Y 608.544,Z 304.015,A -85,B 0,C 180,E1 -432.356,E2 -432.356} C_VEL
LIN {X 0,Y 608.514,Z 330.26,A -85,B 0,C 180,E1 -435.283,E2 -435.283} C_VEL
LIN {X 0,Y 608.506,Z 345.581,A -85,B 0,C 180,E1 -436.966,E2 -436.966} C_VEL
LIN {X 0,Y 608.526,Z 455.075,A -85,B 0,C 180,E1 -438.279,E2 -438.279} C_VEL
LIN {X 0,Y 608.496,Z 468.307,A -85,B 0,C 180,E1 -438.574,E2 -438.574} C_VEL
LIN {X 0,Y 608.509,Z 480.621,A -85,B 0,C 180,E1 -438.982,E2 -438.982} C_VEL
LIN {X 0,Y 608.505,Z 492.681,A -85,B 0,C 180,E1 -439.522,E2 -439.522} C_VEL
LIN {X 0,Y 608.462,Z 504.174,A -85,B 0,C 180,E1 -440.193,E2 -440.193} C_VEL
LIN {X 0,Y 608.471,Z 513.498,A -85,B 0,C 180,E1 -440.864,E2 -440.864} C_VEL
LIN {X 0,Y 608.486,Z 521.318,A -85,B 0,C 180,E1 -441.534,E2 -441.534} C_VEL
LIN {X 0,Y 608.469,Z 529.429,A -85,B 0,C 180,E1 -442.369,E2 -442.369} C_VEL
LIN {X 0,Y 608.439,Z 537.485,A -85,B 0,C 180,E1 -443.369,E2 -443.369} C_VEL
LIN {X 0,Y 608.448,Z 543.874,A -85,B 0,C 180,E1 -444.367,E2 -444.367} C_VEL
LIN {X 0,Y 608.431,Z 548.957,A -85,B 0,C 180,E1 -445.364,E2 -445.364} C_VEL
LIN {X 0,Y 608.448,Z 552.9,A -85,B 0,C 180,E1 -446.359,E2 -446.359} C_VEL
LIN {X 0,Y 608.425,Z 555.811,A -85,B 0,C 180,E1 -447.353,E2 -447.353} C_VEL
LIN {X 0,Y 608.441,Z 557.204,A -85,B 0,C 180,E1 -448.016,E2 -448.016} C_VEL
LIN {X 0,Y 608.447,Z 558.185,A -85,B 0,C 180,E1 -448.678,E2 -448.678} C_VEL
LIN {X 0,Y 608.428,Z 559,A -85,B 0,C 180,E1 -450.001,E2 -450.001} C_VEL
LIN {X 0,Y 608.447,Z 558.182,A -85,B 0,C 180,E1 -451.325,E2 -451.325} C_VEL
LIN {X 0,Y 608.441,Z 557.199,A -85,B 0,C 180,E1 -451.987,E2 -451.987} C_VEL
LIN {X 0,Y 608.425,Z 555.805,A -85,B 0,C 180,E1 -452.649,E2 -452.649} C_VEL
LIN {X 0,Y 608.449,Z 552.891,A -85,B 0,C 180,E1 -453.643,E2 -453.643} C_VEL
LIN {X 0,Y 608.432,Z 548.946,A -85,B 0,C 180,E1 -454.639,E2 -454.639} C_VEL
LIN {X 0,Y 608.448,Z 543.859,A -85,B 0,C 180,E1 -455.635,E2 -455.635} C_VEL
LIN {X 0,Y 608.439,Z 537.465,A -85,B 0,C 180,E1 -456.634,E2 -456.634} C_VEL
LIN {X 0,Y 608.469,Z 529.406,A -85,B 0,C 180,E1 -457.634,E2 -457.634} C_VEL
LIN {X 0,Y 608.473,Z 519.531,A -85,B 0,C 180,E1 -458.636,E2 -458.636} C_VEL
LIN {X 0,Y 608.476,Z 509.005,A -85,B 0,C 180,E1 -459.474,E2 -459.474} C_VEL
LIN {X 0,Y 608.463,Z 498.75,A -85,B 0,C 180,E1 -460.146,E2 -460.146} C_VEL
LIN {X 0,Y 608.517,Z 487.563,A -85,B 0,C 180,E1 -460.726,E2 -460.726} C_VEL
LIN {X 0,Y 608.513,Z 475.871,A -85,B 0,C 180,E1 -461.193,E2 -461.193} C_VEL
LIN {X 0,Y 608.524,Z 463.258,A -85,B 0,C 180,E1 -461.555,E2 -461.555} C_VEL
LIN {X 0,Y 608.529,Z 450.589,A -85,B 0,C 180,E1 -461.787,E2 -461.787} C_VEL
LIN {X 0,Y 608.505,Z 345.48,A -85,B 0,C 180,E1 -463.037,E2 -463.037} C_VEL
LIN {X 0,Y 608.528,Z 319.428,A -85,B 0,C 180,E1 -465.92,E2 -465.92} C_VEL
LIN {X 0,Y 608.565,Z 295.344,A -85,B 0,C 180,E1 -468.621,E2 -468.621} C_VEL
LIN {X 0,Y 608.599,Z 271.57,A -85,B 0,C 180,E1 -471.33,E2 -471.33} C_VEL
LIN {X 0,Y 608.385,Z 264.697,A -85,B 0,C 180,E1 -472.14,E2 -472.14} C_VEL
LIN {X 0,Y 608.403,Z 264.694,A -85,B 0,C 180,E1 -474.572,E2 -474.572} C_VEL
LIN {X 0,Y 608.459,Z 264.695,A -85,B 0,C 180,E1 -477.204,E2 -477.204} C_VEL
LIN {X 0,Y 608.429,Z 264.692,A -85,B 0,C 180,E1 -479.966,E2 -479.966} C_VEL
LIN {X 0,Y 608.414,Z 264.691,A -85,B 0,C 180,E1 -482.516,E2 -482.516} C_VEL
LIN {X 0,Y 608.406,Z 264.694,A -85,B 0,C 180,E1 -484.9,E2 -484.9} C_VEL
LIN {X 0,Y 608.439,Z 264.691,A -85,B 0,C 180,E1 -487.155,E2 -487.155} C_VEL
LIN {X 0,Y 608.461,Z 264.692,A -85,B 0,C 180,E1 -489.437,E2 -489.437} C_VEL
LIN {X 0,Y 608.471,Z 264.687,A -85,B 0,C 180,E1 -492.336,E2 -492.336} C_VEL
LIN {X 0,Y 608.432,Z 264.689,A -85,B 0,C 180,E1 -494.794,E2 -494.794} C_VEL
LIN {X 0,Y 608.434,Z 264.689,A -85,B 0,C 180,E1 -497.039,E2 -497.039} C_VEL
LIN {X 0,Y 608.441,Z 264.694,A -85,B 0,C 180,E1 -499.696,E2 -499.696} C_VEL
LIN {X 0,Y 608.462,Z 264.693,A -85,B 0,C 180,E1 -502.254,E2 -502.254} C_VEL
LIN {X 0,Y 608.473,Z 264.684,A -85,B 0,C 180,E1 -505.085,E2 -505.085} C_VEL
LIN {X 0,Y 608.456,Z 264.691,A -85,B 0,C 180,E1 -507.905,E2 -507.905} C_VEL
LIN {X 0,Y 608.471,Z 264.694,A -85,B 0,C 180,E1 -510.221,E2 -510.221} C_VEL
LIN {X 0,Y 608.46,Z 264.69,A -85,B 0,C 180,E1 -512.788,E2 -512.788} C_VEL
LIN {X 0,Y 608.441,Z 264.688,A -85,B 0,C 180,E1 -515.429,E2 -515.429} C_VEL
LIN {X 0,Y 608.473,Z 264.691,A -85,B 0,C 180,E1 -518.309,E2 -518.309} C_VEL
LIN {X 0,Y 608.437,Z 264.69,A -85,B 0,C 180,E1 -521.281,E2 -521.281} C_VEL
LIN {X 0,Y 608.466,Z 264.685,A -85,B 0,C 180,E1 -523.907,E2 -523.907} C_VEL
LIN {X 0,Y 608.468,Z 264.693,A -85,B 0,C 180,E1 -526.644,E2 -526.644} C_VEL
LIN {X 0,Y 608.431,Z 264.693,A -85,B 0,C 180,E1 -529.35,E2 -529.35} C_VEL
LIN {X 0,Y 608.421,Z 264.694,A -85,B 0,C 180,E1 -531.364,E2 -531.364} C_VEL
LIN {X 0,Y 608.434,Z 264.694,A -85,B 0,C 180,E1 -533.367,E2 -533.367} C_VEL
LIN {X 0,Y 608.424,Z 264.696,A -85,B 0,C 180,E1 -535.362,E2 -535.362} C_VEL
LIN {X 0,Y 608.451,Z 264.695,A -85,B 0,C 180,E1 -537.352,E2 -537.352} C_VEL
LIN {X 0,Y 608.429,Z 264.773,A -85,B 0,C 180,E1 -538.449,E2 -538.449} C_VEL
LIN {X 0,Y 608.537,Z 280.93,A -85,B 0,C 180,E1 -540.993,E2 -540.993} C_VEL
LIN {X 0,Y 608.48,Z 299.14,A -85,B 0,C 180,E1 -543.808,E2 -543.808} C_VEL
LIN {X 0,Y 608.427,Z 315.892,A -85,B 0,C 180,E1 -546.364,E2 -546.364} C_VEL
LIN {X 0,Y 608.462,Z 333.199,A -85,B 0,C 180,E1 -548.977,E2 -548.977} C_VEL
LIN {X 0,Y 608.132,Z 335.662,A -85,B 0,C 180,E1 -549.251,E2 -549.251} C_VEL
LIN {X 0,Y 607.076,Z 339.526,A -85,B 0,C 180,E1 -549.508,E2 -549.508} C_VEL
LIN {X 0,Y 605.643,Z 343.871,A -85,B 0,C 180,E1 -549.683,E2 -549.683} C_VEL
LIN {X 0,Y 603.774,Z 349.576,A -85,B 0,C 180,E1 -549.813,E2 -549.813} C_VEL
LIN {X 0,Y 601.861,Z 357.627,A -85,B 0,C 180,E1 -549.916,E2 -549.916} C_VEL
LIN {X 0,Y 601.531,Z 361.749,A -85,B 0,C 180,E1 -549.961,E2 -549.961} C_VEL
LIN {X 0,Y 601.495,Z 416.181,A -85,B 0,C 180,E1 -550.626,E2 -550.626} C_VEL
LIN {X 0,Y 601.471,Z 425.901,A -85,B 0,C 180,E1 -550.837,E2 -550.837} C_VEL
LIN {X 0,Y 601.47,Z 436.557,A -85,B 0,C 180,E1 -551.183,E2 -551.183} C_VEL
LIN {X 0,Y 601.474,Z 447.936,A -85,B 0,C 180,E1 -551.714,E2 -551.714} C_VEL
LIN {X 0,Y 601.401,Z 456.423,A -85,B 0,C 180,E1 -552.229,E2 -552.229} C_VEL
LIN {X 0,Y 601.395,Z 464.415,A -85,B 0,C 180,E1 -552.829,E2 -552.829} C_VEL
LIN {X 0,Y 601.396,Z 471.888,A -85,B 0,C 180,E1 -553.517,E2 -553.517} C_VEL
LIN {X 0,Y 601.377,Z 479.47,A -85,B 0,C 180,E1 -554.38,E2 -554.38} C_VEL
LIN {X 0,Y 601.368,Z 485.376,A -85,B 0,C 180,E1 -555.246,E2 -555.246} C_VEL
LIN {X 0,Y 601.361,Z 489.253,A -85,B 0,C 180,E1 -555.941,E2 -555.941} C_VEL
LIN {X 0,Y 601.345,Z 492.275,A -85,B 0,C 180,E1 -556.61,E2 -556.61} C_VEL
LIN {X 0,Y 601.326,Z 495.856,A -85,B 0,C 180,E1 -557.691,E2 -557.691} C_VEL
LIN {X 0,Y 601.32,Z 497.487,A -85,B 0,C 180,E1 -558.395,E2 -558.395} C_VEL
LIN {X 0,Y 601.309,Z 498.491,A -85,B 0,C 180,E1 -559.103,E2 -559.103} C_VEL
LIN {X 0,Y 601.308,Z 498.917,A -85,B 0,C 180,E1 -559.813,E2 -559.813} C_VEL
LIN {X 0,Y 601.354,Z 498.677,A -85,B 0,C 180,E1 -560.79,E2 -560.79} C_VEL
LIN {X 0,Y 601.339,Z 496.898,A -85,B 0,C 180,E1 -561.962,E2 -561.962} C_VEL
LIN {X 0,Y 601.357,Z 495.064,A -85,B 0,C 180,E1 -562.686,E2 -562.686} C_VEL
LIN {X 0,Y 601.361,Z 492.55,A -85,B 0,C 180,E1 -563.413,E2 -563.413} C_VEL
LIN {X 0,Y 601.366,Z 488.551,A -85,B 0,C 180,E1 -564.287,E2 -564.287} C_VEL
LIN {X 0,Y 601.371,Z 482.725,A -85,B 0,C 180,E1 -565.25,E2 -565.25} C_VEL
LIN {X 0,Y 601.388,Z 476.564,A -85,B 0,C 180,E1 -566.058,E2 -566.058} C_VEL
LIN {X 0,Y 601.392,Z 470.219,A -85,B 0,C 180,E1 -566.739,E2 -566.739} C_VEL
LIN {X 0,Y 601.397,Z 462.37,A -85,B 0,C 180,E1 -567.431,E2 -567.431} C_VEL
LIN {X 0,Y 601.452,Z 451.904,A -85,B 0,C 180,E1 -568.151,E2 -568.151} C_VEL
LIN {X 0,Y 601.468,Z 442.971,A -85,B 0,C 180,E1 -568.625,E2 -568.625} C_VEL
LIN {X 0,Y 601.477,Z 434.329,A -85,B 0,C 180,E1 -568.985,E2 -568.985} C_VEL
LIN {X 0,Y 601.498,Z 424.99,A -85,B 0,C 180,E1 -569.275,E2 -569.275} C_VEL
LIN {X 0,Y 601.476,Z 416.286,A -85,B 0,C 180,E1 -569.463,E2 -569.463} C_VEL
LIN {X 0,Y 601.399,Z 338.712,A -85,B 0,C 180,E1 -570.408,E2 -570.408} C_VEL
LIN {X 0,Y 601.42,Z 319.637,A -85,B 0,C 180,E1 -573.314,E2 -573.314} C_VEL
LIN {X 0,Y 601.471,Z 302.134,A -85,B 0,C 180,E1 -576.011,E2 -576.011} C_VEL
LIN {X 0,Y 601.502,Z 286.288,A -85,B 0,C 180,E1 -578.484,E2 -578.484} C_VEL
LIN {X 0,Y 601.598,Z 268.912,A -85,B 0,C 180,E1 -581.235,E2 -581.235} C_VEL
LIN {X 0,Y 601.39,Z 265.57,A -85,B 0,C 180,E1 -581.797,E2 -581.797} C_VEL
LIN {X 0,Y 601.38,Z 265.569,A -85,B 0,C 180,E1 -584.535,E2 -584.535} C_VEL
LIN {X 0,Y 601.434,Z 265.57,A -85,B 0,C 180,E1 -587.408,E2 -587.408} C_VEL
LIN {X 0,Y 601.386,Z 265.568,A -85,B 0,C 180,E1 -590.006,E2 -590.006} C_VEL
LIN {X 0,Y 601.386,Z 265.566,A -85,B 0,C 180,E1 -592.625,E2 -592.625} C_VEL
LIN {X 0,Y 601.368,Z 265.57,A -85,B 0,C 180,E1 -595.067,E2 -595.067} C_VEL
LIN {X 0,Y 601.403,Z 265.569,A -85,B 0,C 180,E1 -597.485,E2 -597.485} C_VEL
LIN {X 0,Y 601.403,Z 265.573,A -85,B 0,C 180,E1 -599.857,E2 -599.857} C_VEL
LIN {X 0,Y 601.401,Z 265.565,A -85,B 0,C 180,E1 -602.888,E2 -602.888} C_VEL
LIN {X 0,Y 601.377,Z 265.567,A -85,B 0,C 180,E1 -605.121,E2 -605.121} C_VEL
LIN {X 0,Y 601.378,Z 265.571,A -85,B 0,C 180,E1 -608.04,E2 -608.04} C_VEL
LIN {X 0,Y 601.408,Z 265.57,A -85,B 0,C 180,E1 -610.901,E2 -610.901} C_VEL
LIN {X 0,Y 601.399,Z 265.564,A -85,B 0,C 180,E1 -613.712,E2 -613.712} C_VEL
LIN {X 0,Y 601.384,Z 265.57,A -85,B 0,C 180,E1 -616.483,E2 -616.483} C_VEL
LIN {X 0,Y 601.419,Z 265.572,A -85,B 0,C 180,E1 -619.224,E2 -619.224} C_VEL
LIN {X 0,Y 601.39,Z 265.567,A -85,B 0,C 180,E1 -621.938,E2 -621.938} C_VEL
LIN {X 0,Y 601.38,Z 265.569,A -85,B 0,C 180,E1 -623.962,E2 -623.962} C_VEL
LIN {X 0,Y 601.383,Z 265.57,A -85,B 0,C 180,E1 -625.978,E2 -625.978} C_VEL
LIN {X 0,Y 601.417,Z 265.567,A -85,B 0,C 180,E1 -627.99,E2 -627.99} C_VEL
LIN {X 0,Y 601.362,Z 265.569,A -85,B 0,C 180,E1 -630.668,E2 -630.668} C_VEL
LIN {X 0,Y 601.4,Z 265.565,A -85,B 0,C 180,E1 -632.678,E2 -632.678} C_VEL
LIN {X 0,Y 601.379,Z 265.568,A -85,B 0,C 180,E1 -635.363,E2 -635.363} C_VEL
LIN {X 0,Y 601.4,Z 265.574,A -85,B 0,C 180,E1 -638.059,E2 -638.059} C_VEL
LIN {X 0,Y 601.401,Z 265.566,A -85,B 0,C 180,E1 -640.998,E2 -640.998} C_VEL
LIN {X 0,Y 601.371,Z 265.568,A -85,B 0,C 180,E1 -643.514,E2 -643.514} C_VEL
LIN {X 0,Y 601.407,Z 265.568,A -85,B 0,C 180,E1 -646.285,E2 -646.285} C_VEL
LIN {X 0,Y 601.4,Z 265.571,A -85,B 0,C 180,E1 -649.096,E2 -649.096} C_VEL
LIN {X 0,Y 601.385,Z 265.573,A -85,B 0,C 180,E1 -651.236,E2 -651.236} C_VEL
LIN {X 0,Y 601.369,Z 265.574,A -85,B 0,C 180,E1 -653.408,E2 -653.408} C_VEL
LIN {X 0,Y 601.381,Z 265.568,A -85,B 0,C 180,E1 -655.86,E2 -655.86} C_VEL
LIN {X 0,Y 601.368,Z 265.571,A -85,B 0,C 180,E1 -657.865,E2 -657.865} C_VEL
LIN {X 0,Y 601.382,Z 265.568,A -85,B 0,C 180,E1 -660.162,E2 -660.162} C_VEL
LIN {X 0,Y 601.372,Z 265.568,A -85,B 0,C 180,E1 -662.707,E2 -662.707} C_VEL
LIN {X 0,Y 601.351,Z 265.572,A -85,B 0,C 180,E1 -665.105,E2 -665.105} C_VEL
LIN {X 0,Y 601.403,Z 265.567,A -85,B 0,C 180,E1 -667.415,E2 -667.415} C_VEL
LIN {X 0,Y 601.38,Z 265.579,A -85,B 0,C 180,E1 -669.991,E2 -669.991} C_VEL
LIN {X 0,Y 601.409,Z 265.566,A -85,B 0,C 180,E1 -672.663,E2 -672.663} C_VEL
LIN {X 0,Y 601.361,Z 265.569,A -85,B 0,C 180,E1 -675.475,E2 -675.475} C_VEL
LIN {X 0,Y 601.393,Z 265.572,A -85,B 0,C 180,E1 -678.232,E2 -678.232} C_VEL
LIN {X 0,Y 601.4,Z 265.572,A -85,B 0,C 180,E1 -680.872,E2 -680.872} C_VEL
LIN {X 0,Y 601.375,Z 265.567,A -85,B 0,C 180,E1 -683.733,E2 -683.733} C_VEL
LIN {X 0,Y 601.367,Z 265.568,A -85,B 0,C 180,E1 -686.063,E2 -686.063} C_VEL
LIN {X 0,Y 601.39,Z 265.568,A -85,B 0,C 180,E1 -688.538,E2 -688.538} C_VEL
LIN {X 0,Y 601.419,Z 265.572,A -85,B 0,C 180,E1 -691.372,E2 -691.372} C_VEL
LIN {X 0,Y 601.356,Z 265.571,A -85,B 0,C 180,E1 -694.129,E2 -694.129} C_VEL
LIN {X 0,Y 601.365,Z 265.568,A -85,B 0,C 180,E1 -696.587,E2 -696.587} C_VEL
LIN {X 0,Y 601.395,Z 265.572,A -85,B 0,C 180,E1 -699.477,E2 -699.477} C_VEL
LIN {X 0,Y 601.357,Z 265.574,A -85,B 0,C 180,E1 -702.31,E2 -702.31} C_VEL
LIN {X 0,Y 601.379,Z 265.571,A -85,B 0,C 180,E1 -704.407,E2 -704.407} C_VEL
LIN {X 0,Y 601.377,Z 265.572,A -85,B 0,C 180,E1 -706.483,E2 -706.483} C_VEL
LIN {X 0,Y 601.346,Z 265.571,A -85,B 0,C 180,E1 -709.222,E2 -709.222} C_VEL
LIN {X 0,Y 601.386,Z 265.569,A -85,B 0,C 180,E1 -711.938,E2 -711.938} C_VEL
LIN {X 0,Y 601.432,Z 265.572,A -85,B 0,C 180,E1 -714.636,E2 -714.636} C_VEL
LIN {X 0,Y 601.385,Z 265.568,A -85,B 0,C 180,E1 -717.32,E2 -717.32} C_VEL
LIN {X 0,Y 601.367,Z 265.568,A -85,B 0,C 180,E1 -720,E2 -720} C_VEL
LIN {X 0,Y 601.392,Z 265.57,A -85,B 0,C 180,E1 -722.679,E2 -722.679} C_VEL
LIN {X 0,Y 601.432,Z 265.569,A -85,B 0,C 180,E1 -725.364,E2 -725.364} C_VEL
LIN {X 0,Y 601.377,Z 265.568,A -85,B 0,C 180,E1 -728.061,E2 -728.061} C_VEL
LIN {X 0,Y 601.344,Z 265.572,A -85,B 0,C 180,E1 -730.777,E2 -730.777} C_VEL
LIN {X 0,Y 601.377,Z 265.576,A -85,B 0,C 180,E1 -733.516,E2 -733.516} C_VEL
LIN {X 0,Y 601.402,Z 265.568,A -85,B 0,C 180,E1 -736.288,E2 -736.288} C_VEL
LIN {X 0,Y 601.354,Z 265.57,A -85,B 0,C 180,E1 -739.101,E2 -739.101} C_VEL
LIN {X 0,Y 601.345,Z 265.571,A -85,B 0,C 180,E1 -741.241,E2 -741.241} C_VEL
LIN {X 0,Y 601.36,Z 265.57,A -85,B 0,C 180,E1 -743.412,E2 -743.412} C_VEL
LIN {X 0,Y 601.355,Z 265.573,A -85,B 0,C 180,E1 -745.871,E2 -745.871} C_VEL
LIN {X 0,Y 601.408,Z 265.57,A -85,B 0,C 180,E1 -748.797,E2 -748.797} C_VEL
LIN {X 0,Y 601.342,Z 265.571,A -85,B 0,C 180,E1 -751.73,E2 -751.73} C_VEL
LIN {X 0,Y 601.371,Z 265.569,A -85,B 0,C 180,E1 -754.122,E2 -754.122} C_VEL
LIN {X 0,Y 601.371,Z 265.572,A -85,B 0,C 180,E1 -756.585,E2 -756.585} C_VEL
LIN {X 0,Y 601.395,Z 265.57,A -85,B 0,C 180,E1 -759.539,E2 -759.539} C_VEL
LIN {X 0,Y 601.371,Z 265.571,A -85,B 0,C 180,E1 -761.769,E2 -761.769} C_VEL
LIN {X 0,Y 601.407,Z 265.572,A -85,B 0,C 180,E1 -763.588,E2 -763.588} C_VEL
LIN {X 0,Y 601.361,Z 265.569,A -85,B 0,C 180,E1 -766.434,E2 -766.434} C_VEL
LIN {X 0,Y 601.365,Z 265.569,A -85,B 0,C 180,E1 -768.413,E2 -768.413} C_VEL
LIN {X 0,Y 601.345,Z 265.571,A -85,B 0,C 180,E1 -770.875,E2 -770.875} C_VEL
LIN {X 0,Y 601.353,Z 265.573,A -85,B 0,C 180,E1 -773.419,E2 -773.419} C_VEL
LIN {X 0,Y 601.398,Z 265.576,A -85,B 0,C 180,E1 -776.069,E2 -776.069} C_VEL
LIN {X 0,Y 601.356,Z 265.57,A -85,B 0,C 180,E1 -779.059,E2 -779.059} C_VEL
LIN {X 0,Y 601.332,Z 265.573,A -85,B 0,C 180,E1 -781.373,E2 -781.373} C_VEL
LIN {X 0,Y 601.345,Z 265.572,A -85,B 0,C 180,E1 -783.638,E2 -783.638} C_VEL
LIN {X 0,Y 601.365,Z 265.57,A -85,B 0,C 180,E1 -785.86,E2 -785.86} C_VEL
LIN {X 0,Y 601.377,Z 265.725,A -85,B 0,C 180,E1 -787.718,E2 -787.718} C_VEL
LIN {X 0,Y 601.691,Z 270.051,A -85,B 0,C 180,E1 -788.236,E2 -788.236} C_VEL
LIN {X 0,Y 601.644,Z 293.208,A -85,B 0,C 180,E1 -790.912,E2 -790.912} C_VEL
LIN {X 0,Y 601.549,Z 315.669,A -85,B 0,C 180,E1 -793.466,E2 -793.466} C_VEL
LIN {X 0,Y 601.497,Z 340.204,A -85,B 0,C 180,E1 -796.22,E2 -796.22} C_VEL
LIN {X 0,Y 601.497,Z 345.581,A -85,B 0,C 180,E1 -796.811,E2 -796.811} C_VEL
LIN {X 0,Y 601.597,Z 455.017,A -85,B 0,C 180,E1 -798.142,E2 -798.142} C_VEL
LIN {X 0,Y 601.551,Z 467.548,A -85,B 0,C 180,E1 -798.419,E2 -798.419} C_VEL
LIN {X 0,Y 601.547,Z 481.004,A -85,B 0,C 180,E1 -798.867,E2 -798.867} C_VEL
LIN {X 0,Y 601.516,Z 492.679,A -85,B 0,C 180,E1 -799.398,E2 -799.398} C_VEL
LIN {X 0,Y 601.461,Z 504.176,A -85,B 0,C 180,E1 -800.078,E2 -800.078} C_VEL
LIN {X 0,Y 601.43,Z 513.5,A -85,B 0,C 180,E1 -800.756,E2 -800.756} C_VEL
LIN {X 0,Y 601.421,Z 521.317,A -85,B 0,C 180,E1 -801.434,E2 -801.434} C_VEL
LIN {X 0,Y 601.389,Z 529.429,A -85,B 0,C 180,E1 -802.279,E2 -802.279} C_VEL
LIN {X 0,Y 601.375,Z 537.475,A -85,B 0,C 180,E1 -803.291,E2 -803.291} C_VEL
LIN {X 0,Y 601.37,Z 543.864,A -85,B 0,C 180,E1 -804.301,E2 -804.301} C_VEL
LIN {X 0,Y 601.336,Z 548.951,A -85,B 0,C 180,E1 -805.309,E2 -805.309} C_VEL
LIN {X 0,Y 601.367,Z 552.891,A -85,B 0,C 180,E1 -806.316,E2 -806.316} C_VEL
LIN {X 0,Y 601.325,Z 555.801,A -85,B 0,C 180,E1 -807.322,E2 -807.322} C_VEL
LIN {X 0,Y 601.34,Z 557.202,A -85,B 0,C 180,E1 -807.992,E2 -807.992} C_VEL
LIN {X 0,Y 601.347,Z 558.186,A -85,B 0,C 180,E1 -808.662,E2 -808.662} C_VEL
LIN {X 0,Y 601.329,Z 559,A -85,B 0,C 180,E1 -810.001,E2 -810.001} C_VEL
LIN {X 0,Y 601.347,Z 558.183,A -85,B 0,C 180,E1 -811.341,E2 -811.341} C_VEL
LIN {X 0,Y 601.34,Z 557.198,A -85,B 0,C 180,E1 -812.01,E2 -812.01} C_VEL
LIN {X 0,Y 601.325,Z 555.795,A -85,B 0,C 180,E1 -812.681,E2 -812.681} C_VEL
LIN {X 0,Y 601.367,Z 552.882,A -85,B 0,C 180,E1 -813.686,E2 -813.686} C_VEL
LIN {X 0,Y 601.336,Z 548.939,A -85,B 0,C 180,E1 -814.694,E2 -814.694} C_VEL
LIN {X 0,Y 601.37,Z 543.849,A -85,B 0,C 180,E1 -815.702,E2 -815.702} C_VEL
LIN {X 0,Y 601.378,Z 537.456,A -85,B 0,C 180,E1 -816.712,E2 -816.712} C_VEL
LIN {X 0,Y 601.39,Z 529.406,A -85,B 0,C 180,E1 -817.724,E2 -817.724} C_VEL
LIN {X 0,Y 601.432,Z 519.531,A -85,B 0,C 180,E1 -818.738,E2 -818.738} C_VEL
LIN {X 0,Y 601.468,Z 509.008,A -85,B 0,C 180,E1 -819.585,E2 -819.585} C_VEL
LIN {X 0,Y 601.462,Z 498.752,A -85,B 0,C 180,E1 -820.265,E2 -820.265} C_VEL
LIN {X 0,Y 601.535,Z 487.873,A -85,B 0,C 180,E1 -820.837,E2 -820.837} C_VEL
LIN {X 0,Y 601.543,Z 476.451,A -85,B 0,C 180,E1 -821.303,E2 -821.303} C_VEL
LIN {X 0,Y 601.564,Z 464.171,A -85,B 0,C 180,E1 -821.669,E2 -821.669} C_VEL
LIN {X 0,Y 601.596,Z 450.589,A -85,B 0,C 180,E1 -821.925,E2 -821.925} C_VEL
LIN {X 0,Y 601.573,Z 346.243,A -85,B 0,C 180,E1 -823.179,E2 -823.179} C_VEL
LIN {X 0,Y 601.487,Z 345.287,A -85,B 0,C 180,E1 -823.213,E2 -823.213} C_VEL
LIN {X 0,Y 601.547,Z 320.972,A -85,B 0,C 180,E1 -825.935,E2 -825.935} C_VEL
LIN {X 0,Y 601.654,Z 296.098,A -85,B 0,C 180,E1 -828.757,E2 -828.757} C_VEL
LIN {X 0,Y 601.707,Z 271.57,A -85,B 0,C 180,E1 -831.587,E2 -831.587} C_VEL
LIN {X 0,Y 601.473,Z 266.26,A -85,B 0,C 180,E1 -832.216,E2 -832.216} C_VEL
LIN {X 0,Y 601.35,Z 265.576,A -85,B 0,C 180,E1 -832.308,E2 -832.308} C_VEL
LIN {X 0,Y 601.369,Z 265.574,A -85,B 0,C 180,E1 -834.879,E2 -834.879} C_VEL
LIN {X 0,Y 601.395,Z 265.578,A -85,B 0,C 180,E1 -837.359,E2 -837.359} C_VEL
LIN {X 0,Y 601.389,Z 265.568,A -85,B 0,C 180,E1 -840.164,E2 -840.164} C_VEL
LIN {X 0,Y 601.383,Z 265.568,A -85,B 0,C 180,E1 -842.71,E2 -842.71} C_VEL
LIN {X 0,Y 601.37,Z 265.572,A -85,B 0,C 180,E1 -845.109,E2 -845.109} C_VEL
LIN {X 0,Y 601.417,Z 265.57,A -85,B 0,C 180,E1 -847.418,E2 -847.418} C_VEL
LIN {X 0,Y 601.402,Z 265.571,A -85,B 0,C 180,E1 -849.993,E2 -849.993} C_VEL
LIN {X 0,Y 601.418,Z 265.563,A -85,B 0,C 180,E1 -852.666,E2 -852.666} C_VEL
LIN {X 0,Y 601.404,Z 265.569,A -85,B 0,C 180,E1 -855.48,E2 -855.48} C_VEL
LIN {X 0,Y 601.418,Z 265.567,A -85,B 0,C 180,E1 -858.403,E2 -858.403} C_VEL
LIN {X 0,Y 601.426,Z 265.562,A -85,B 0,C 180,E1 -860.875,E2 -860.875} C_VEL
LIN {X 0,Y 601.425,Z 265.566,A -85,B 0,C 180,E1 -863.731,E2 -863.731} C_VEL
LIN {X 0,Y 601.42,Z 265.571,A -85,B 0,C 180,E1 -866.06,E2 -866.06} C_VEL
LIN {X 0,Y 601.418,Z 265.569,A -85,B 0,C 180,E1 -868.539,E2 -868.539} C_VEL
LIN {X 0,Y 601.426,Z 265.562,A -85,B 0,C 180,E1 -871.373,E2 -871.373} C_VEL
LIN {X 0,Y 601.413,Z 265.569,A -85,B 0,C 180,E1 -874.124,E2 -874.124} C_VEL
LIN {X 0,Y 601.406,Z 265.574,A -85,B 0,C 180,E1 -876.59,E2 -876.59} C_VEL
LIN {X 0,Y 601.408,Z 265.566,A -85,B 0,C 180,E1 -879.196,E2 -879.196} C_VEL
LIN {X 0,Y 601.403,Z 265.565,A -85,B 0,C 180,E1 -881.608,E2 -881.608} C_VEL
LIN {X 0,Y 601.415,Z 265.569,A -85,B 0,C 180,E1 -884.409,E2 -884.409} C_VEL
LIN {X 0,Y 601.398,Z 265.57,A -85,B 0,C 180,E1 -887.172,E2 -887.172} C_VEL
LIN {X 0,Y 601.403,Z 265.565,A -85,B 0,C 180,E1 -889.905,E2 -889.905} C_VEL
LIN {X 0,Y 601.431,Z 265.566,A -85,B 0,C 180,E1 -892.615,E2 -892.615} C_VEL
LIN {X 0,Y 601.395,Z 265.573,A -85,B 0,C 180,E1 -895.308,E2 -895.308} C_VEL
LIN {X 0,Y 601.416,Z 265.572,A -85,B 0,C 180,E1 -897.321,E2 -897.321} C_VEL
LIN {X 0,Y 601.415,Z 265.657,A -85,B 0,C 180,E1 -898.326,E2 -898.326} C_VEL
LIN {X 0,Y 601.509,Z 275.069,A -85,B 0,C 180,E1 -899.833,E2 -899.833} C_VEL
LIN {X 0,Y 601.506,Z 290.994,A -85,B 0,C 180,E1 -902.344,E2 -902.344} C_VEL
LIN {X 0,Y 601.463,Z 309.357,A -85,B 0,C 180,E1 -905.196,E2 -905.196} C_VEL
LIN {X 0,Y 601.39,Z 326.948,A -85,B 0,C 180,E1 -907.893,E2 -907.893} C_VEL
LIN {X 0,Y 601.397,Z 338.641,A -85,B 0,C 180,E1 -909.671,E2 -909.671} C_VEL
LIN {X 0,Y 601.531,Z 361.749,A -85,B 0,C 180,E1 -909.961,E2 -909.961} C_VEL
LIN {X 0,Y 600.843,Z 367.594,A -85,B 0,C 180,E1 -910.019,E2 -910.019} C_VEL
LIN {X 0,Y 595.18,Z 386.57,A -85,B 0,C 180,E1 -910.15,E2 -910.15} C_VEL
LIN {X 0,Y 594.536,Z 392.413,A -85,B 0,C 180,E1 -910.209,E2 -910.209} C_VEL
LIN {X 0,Y 594.485,Z 417.601,A -85,B 0,C 180,E1 -910.537,E2 -910.537} C_VEL
LIN {X 0,Y 594.461,Z 429.221,A -85,B 0,C 180,E1 -910.818,E2 -910.818} C_VEL
LIN {X 0,Y 594.419,Z 439.407,A -85,B 0,C 180,E1 -911.198,E2 -911.198} C_VEL
LIN {X 0,Y 594.415,Z 449.116,A -85,B 0,C 180,E1 -911.682,E2 -911.682} C_VEL
LIN {X 0,Y 594.364,Z 457.378,A -85,B 0,C 180,E1 -912.203,E2 -912.203} C_VEL
LIN {X 0,Y 594.339,Z 465.215,A -85,B 0,C 180,E1 -912.81,E2 -912.81} C_VEL
LIN {X 0,Y 594.31,Z 474.228,A -85,B 0,C 180,E1 -913.681,E2 -913.681} C_VEL
LIN {X 0,Y 594.31,Z 481.179,A -85,B 0,C 180,E1 -914.554,E2 -914.554} C_VEL
LIN {X 0,Y 594.288,Z 484.758,A -85,B 0,C 180,E1 -915.081,E2 -915.081} C_VEL
LIN {X 0,Y 594.272,Z 488.719,A -85,B 0,C 180,E1 -915.784,E2 -915.784} C_VEL
LIN {X 0,Y 594.252,Z 492.743,A -85,B 0,C 180,E1 -916.688,E2 -916.688} C_VEL
LIN {X 0,Y 594.216,Z 496.44,A -85,B 0,C 180,E1 -917.91,E2 -917.91} C_VEL
LIN {X 0,Y 594.222,Z 498.221,A -85,B 0,C 180,E1 -918.896,E2 -918.896} C_VEL
LIN {X 0,Y 594.211,Z 499,A -85,B 0,C 180,E1 -920.06,E2 -920.06} C_VEL
LIN {X 0,Y 594.257,Z 498.608,A -85,B 0,C 180,E1 -920.897,E2 -920.897} C_VEL
LIN {X 0,Y 594.224,Z 497.784,A -85,B 0,C 180,E1 -921.509,E2 -921.509} C_VEL
LIN {X 0,Y 594.261,Z 495.051,A -85,B 0,C 180,E1 -922.721,E2 -922.721} C_VEL
LIN {X 0,Y 594.271,Z 491.437,A -85,B 0,C 180,E1 -923.709,E2 -923.709} C_VEL
LIN {X 0,Y 594.269,Z 486.863,A -85,B 0,C 180,E1 -924.638,E2 -924.638} C_VEL
LIN {X 0,Y 594.295,Z 482.225,A -85,B 0,C 180,E1 -925.385,E2 -925.385} C_VEL
LIN {X 0,Y 594.318,Z 476.638,A -85,B 0,C 180,E1 -926.121,E2 -926.121} C_VEL
LIN {X 0,Y 594.33,Z 469.486,A -85,B 0,C 180,E1 -926.892,E2 -926.892} C_VEL
LIN {X 0,Y 594.378,Z 459.897,A -85,B 0,C 180,E1 -927.711,E2 -927.711} C_VEL
LIN {X 0,Y 594.421,Z 450.618,A -85,B 0,C 180,E1 -928.321,E2 -928.321} C_VEL
LIN {X 0,Y 594.463,Z 442.422,A -85,B 0,C 180,E1 -928.753,E2 -928.753} C_VEL
LIN {X 0,Y 594.462,Z 434.342,A -85,B 0,C 180,E1 -929.091,E2 -929.091} C_VEL
LIN {X 0,Y 594.481,Z 425.138,A -85,B 0,C 180,E1 -929.382,E2 -929.382} C_VEL
LIN {X 0,Y 594.478,Z 416.182,A -85,B 0,C 180,E1 -929.576,E2 -929.576} C_VEL
LIN {X 0,Y 594.445,Z 339.717,A -85,B 0,C 180,E1 -930.516,E2 -930.516} C_VEL
LIN {X 0,Y 594.332,Z 338.626,A -85,B 0,C 180,E1 -930.546,E2 -930.546} C_VEL
LIN {X 0,Y 594.379,Z 320.407,A -85,B 0,C 180,E1 -933.355,E2 -933.355} C_VEL
LIN {X 0,Y 594.447,Z 303.257,A -85,B 0,C 180,E1 -936.029,E2 -936.029} C_VEL
LIN {X 0,Y 594.517,Z 286.185,A -85,B 0,C 180,E1 -938.725,E2 -938.725} C_VEL
LIN {X 0,Y 594.63,Z 268.034,A -85,B 0,C 180,E1 -941.638,E2 -941.638} C_VEL
LIN {X 0,Y 594.341,Z 266.449,A -85,B 0,C 180,E1 -941.94,E2 -941.94} C_VEL
LIN {X 0,Y 594.328,Z 266.452,A -85,B 0,C 180,E1 -944.809,E2 -944.809} C_VEL
LIN {X 0,Y 594.377,Z 266.445,A -85,B 0,C 180,E1 -947.629,E2 -947.629} C_VEL
LIN {X 0,Y 594.347,Z 266.443,A -85,B 0,C 180,E1 -950.32,E2 -950.32} C_VEL
LIN {X 0,Y 594.346,Z 266.444,A -85,B 0,C 180,E1 -952.913,E2 -952.913} C_VEL
LIN {X 0,Y 594.358,Z 266.452,A -85,B 0,C 180,E1 -955.865,E2 -955.865} C_VEL
LIN {X 0,Y 594.353,Z 266.443,A -85,B 0,C 180,E1 -958.651,E2 -958.651} C_VEL
LIN {X 0,Y 594.331,Z 266.445,A -85,B 0,C 180,E1 -961.052,E2 -961.052} C_VEL
LIN {X 0,Y 594.349,Z 266.443,A -85,B 0,C 180,E1 -963.3,E2 -963.3} C_VEL
LIN {X 0,Y 594.334,Z 266.445,A -85,B 0,C 180,E1 -965.579,E2 -965.579} C_VEL
LIN {X 0,Y 594.348,Z 266.455,A -85,B 0,C 180,E1 -968.497,E2 -968.497} C_VEL
LIN {X 0,Y 594.347,Z 266.444,A -85,B 0,C 180,E1 -971.382,E2 -971.382} C_VEL
LIN {X 0,Y 594.37,Z 266.441,A -85,B 0,C 180,E1 -973.514,E2 -973.514} C_VEL
LIN {X 0,Y 594.347,Z 266.445,A -85,B 0,C 180,E1 -976.32,E2 -976.32} C_VEL
LIN {X 0,Y 594.379,Z 266.451,A -85,B 0,C 180,E1 -979.094,E2 -979.094} C_VEL
LIN {X 0,Y 594.347,Z 266.445,A -85,B 0,C 180,E1 -981.842,E2 -981.842} C_VEL
LIN {X 0,Y 594.347,Z 266.443,A -85,B 0,C 180,E1 -984.571,E2 -984.571} C_VEL
LIN {X 0,Y 594.387,Z 266.444,A -85,B 0,C 180,E1 -987.288,E2 -987.288} C_VEL
LIN {X 0,Y 594.413,Z 266.441,A -85,B 0,C 180,E1 -989.999,E2 -989.999} C_VEL
LIN {X 0,Y 594.368,Z 266.441,A -85,B 0,C 180,E1 -992.709,E2 -992.709} C_VEL
LIN {X 0,Y 594.349,Z 266.444,A -85,B 0,C 180,E1 -995.426,E2 -995.426} C_VEL
LIN {X 0,Y 594.353,Z 266.454,A -85,B 0,C 180,E1 -998.155,E2 -998.155} C_VEL
LIN {X 0,Y 594.371,Z 266.441,A -85,B 0,C 180,E1 -1001.062,E2 -1001.062} C_VEL
LIN {X 0,Y 594.338,Z 266.444,A -85,B 0,C 180,E1 -1003.677,E2 -1003.677} C_VEL
LIN {X 0,Y 594.388,Z 266.446,A -85,B 0,C 180,E1 -1006.482,E2 -1006.482} C_VEL
LIN {X 0,Y 594.347,Z 266.446,A -85,B 0,C 180,E1 -1009.332,E2 -1009.332} C_VEL
LIN {X 0,Y 594.339,Z 266.446,A -85,B 0,C 180,E1 -1011.501,E2 -1011.501} C_VEL
LIN {X 0,Y 594.329,Z 266.446,A -85,B 0,C 180,E1 -1014.445,E2 -1014.445} C_VEL
LIN {X 0,Y 594.348,Z 266.445,A -85,B 0,C 180,E1 -1016.697,E2 -1016.697} C_VEL
LIN {X 0,Y 594.354,Z 266.446,A -85,B 0,C 180,E1 -1018.995,E2 -1018.995} C_VEL
LIN {X 0,Y 594.354,Z 266.452,A -85,B 0,C 180,E1 -1021.638,E2 -1021.638} C_VEL
LIN {X 0,Y 594.339,Z 266.444,A -85,B 0,C 180,E1 -1024.577,E2 -1024.577} C_VEL
LIN {X 0,Y 594.362,Z 266.447,A -85,B 0,C 180,E1 -1027.604,E2 -1027.604} C_VEL
LIN {X 0,Y 594.352,Z 266.445,A -85,B 0,C 180,E1 -1030.562,E2 -1030.562} C_VEL
LIN {X 0,Y 594.324,Z 266.446,A -85,B 0,C 180,E1 -1033.296,E2 -1033.296} C_VEL
LIN {X 0,Y 594.338,Z 266.452,A -85,B 0,C 180,E1 -1036.156,E2 -1036.156} C_VEL
LIN {X 0,Y 594.342,Z 266.445,A -85,B 0,C 180,E1 -1039.173,E2 -1039.173} C_VEL
LIN {X 0,Y 594.336,Z 266.446,A -85,B 0,C 180,E1 -1042.055,E2 -1042.055} C_VEL
LIN {X 0,Y 594.341,Z 266.452,A -85,B 0,C 180,E1 -1044.667,E2 -1044.667} C_VEL
LIN {X 0,Y 594.331,Z 266.455,A -85,B 0,C 180,E1 -1047.084,E2 -1047.084} C_VEL
LIN {X 0,Y 594.336,Z 266.447,A -85,B 0,C 180,E1 -1049.668,E2 -1049.668} C_VEL
LIN {X 0,Y 594.352,Z 266.445,A -85,B 0,C 180,E1 -1051.771,E2 -1051.771} C_VEL
LIN {X 0,Y 594.321,Z 266.448,A -85,B 0,C 180,E1 -1054.053,E2 -1054.053} C_VEL
LIN {X 0,Y 594.343,Z 266.444,A -85,B 0,C 180,E1 -1056.294,E2 -1056.294} C_VEL
LIN {X 0,Y 594.356,Z 266.445,A -85,B 0,C 180,E1 -1059.222,E2 -1059.222} C_VEL
LIN {X 0,Y 594.338,Z 266.451,A -85,B 0,C 180,E1 -1062.094,E2 -1062.094} C_VEL
LIN {X 0,Y 594.335,Z 266.452,A -85,B 0,C 180,E1 -1064.218,E2 -1064.218} C_VEL
LIN {X 0,Y 594.344,Z 266.451,A -85,B 0,C 180,E1 -1066.32,E2 -1066.32} C_VEL
LIN {X 0,Y 594.305,Z 266.448,A -85,B 0,C 180,E1 -1069.093,E2 -1069.093} C_VEL
LIN {X 0,Y 594.358,Z 266.444,A -85,B 0,C 180,E1 -1071.842,E2 -1071.842} C_VEL
LIN {X 0,Y 594.386,Z 266.45,A -85,B 0,C 180,E1 -1074.572,E2 -1074.572} C_VEL
LIN {X 0,Y 594.352,Z 266.445,A -85,B 0,C 180,E1 -1077.289,E2 -1077.289} C_VEL
LIN {X 0,Y 594.337,Z 266.444,A -85,B 0,C 180,E1 -1080,E2 -1080} C_VEL
LIN {X 0,Y 594.358,Z 266.447,A -85,B 0,C 180,E1 -1082.711,E2 -1082.711} C_VEL
LIN {X 0,Y 594.384,Z 266.446,A -85,B 0,C 180,E1 -1085.427,E2 -1085.427} C_VEL
LIN {X 0,Y 594.352,Z 266.443,A -85,B 0,C 180,E1 -1088.157,E2 -1088.157} C_VEL
LIN {X 0,Y 594.319,Z 266.45,A -85,B 0,C 180,E1 -1091.075,E2 -1091.075} C_VEL
LIN {X 0,Y 594.344,Z 266.456,A -85,B 0,C 180,E1 -1093.679,E2 -1093.679} C_VEL
LIN {X 0,Y 594.327,Z 266.445,A -85,B 0,C 180,E1 -1096.721,E2 -1096.721} C_VEL
LIN {X 0,Y 594.31,Z 266.449,A -85,B 0,C 180,E1 -1099.336,E2 -1099.336} C_VEL
LIN {X 0,Y 594.314,Z 266.449,A -85,B 0,C 180,E1 -1101.505,E2 -1101.505} C_VEL
LIN {X 0,Y 594.341,Z 266.446,A -85,B 0,C 180,E1 -1103.706,E2 -1103.706} C_VEL
LIN {X 0,Y 594.327,Z 266.452,A -85,B 0,C 180,E1 -1106.702,E2 -1106.702} C_VEL
LIN {X 0,Y 594.338,Z 266.448,A -85,B 0,C 180,E1 -1109,E2 -1109} C_VEL
LIN {X 0,Y 594.318,Z 266.446,A -85,B 0,C 180,E1 -1111.645,E2 -1111.645} C_VEL
LIN {X 0,Y 594.356,Z 266.448,A -85,B 0,C 180,E1 -1114.581,E2 -1114.581} C_VEL
LIN {X 0,Y 594.34,Z 266.446,A -85,B 0,C 180,E1 -1117.612,E2 -1117.612} C_VEL
LIN {X 0,Y 594.317,Z 266.448,A -85,B 0,C 180,E1 -1120.571,E2 -1120.571} C_VEL
LIN {X 0,Y 594.329,Z 266.456,A -85,B 0,C 180,E1 -1123.302,E2 -1123.302} C_VEL
LIN {X 0,Y 594.308,Z 266.449,A -85,B 0,C 180,E1 -1126.166,E2 -1126.166} C_VEL
LIN {X 0,Y 594.325,Z 266.446,A -85,B 0,C 180,E1 -1128.538,E2 -1128.538} C_VEL
LIN {X 0,Y 594.335,Z 266.447,A -85,B 0,C 180,E1 -1131.301,E2 -1131.301} C_VEL
LIN {X 0,Y 594.334,Z 266.452,A -85,B 0,C 180,E1 -1133.76,E2 -1133.76} C_VEL
LIN {X 0,Y 594.334,Z 266.454,A -85,B 0,C 180,E1 -1136.241,E2 -1136.241} C_VEL
LIN {X 0,Y 594.331,Z 266.449,A -85,B 0,C 180,E1 -1138.653,E2 -1138.653} C_VEL
LIN {X 0,Y 594.308,Z 266.449,A -85,B 0,C 180,E1 -1141.055,E2 -1141.055} C_VEL
LIN {X 0,Y 594.328,Z 266.447,A -85,B 0,C 180,E1 -1143.302,E2 -1143.302} C_VEL
LIN {X 0,Y 594.31,Z 266.449,A -85,B 0,C 180,E1 -1145.582,E2 -1145.582} C_VEL
LIN {X 0,Y 594.335,Z 266.591,A -85,B 0,C 180,E1 -1147.542,E2 -1147.542} C_VEL
LIN {X 0,Y 594.806,Z 270.051,A -85,B 0,C 180,E1 -1147.97,E2 -1147.97} C_VEL
LIN {X 0,Y 594.739,Z 293.208,A -85,B 0,C 180,E1 -1150.682,E2 -1150.682} C_VEL
LIN {X 0,Y 594.605,Z 316.31,A -85,B 0,C 180,E1 -1153.341,E2 -1153.341} C_VEL
LIN {X 0,Y 594.501,Z 341.429,A -85,B 0,C 180,E1 -1156.193,E2 -1156.193} C_VEL
LIN {X 0,Y 594.487,Z 345.581,A -85,B 0,C 180,E1 -1156.653,E2 -1156.653} C_VEL
LIN {X 0,Y 594.777,Z 352.735,A -85,B 0,C 180,E1 -1156.746,E2 -1156.746} C_VEL
LIN {X 0,Y 594.649,Z 454.951,A -85,B 0,C 180,E1 -1158.001,E2 -1158.001} C_VEL
LIN {X 0,Y 594.596,Z 467.549,A -85,B 0,C 180,E1 -1158.281,E2 -1158.281} C_VEL
LIN {X 0,Y 594.565,Z 480.206,A -85,B 0,C 180,E1 -1158.704,E2 -1158.704} C_VEL
LIN {X 0,Y 594.531,Z 492.678,A -85,B 0,C 180,E1 -1159.272,E2 -1159.272} C_VEL
LIN {X 0,Y 594.448,Z 504.172,A -85,B 0,C 180,E1 -1159.96,E2 -1159.96} C_VEL
LIN {X 0,Y 594.402,Z 513.498,A -85,B 0,C 180,E1 -1160.646,E2 -1160.646} C_VEL
LIN {X 0,Y 594.373,Z 521.316,A -85,B 0,C 180,E1 -1161.331,E2 -1161.331} C_VEL
LIN {X 0,Y 594.34,Z 529.43,A -85,B 0,C 180,E1 -1162.187,E2 -1162.187} C_VEL
LIN {X 0,Y 594.309,Z 537.463,A -85,B 0,C 180,E1 -1163.211,E2 -1163.211} C_VEL
LIN {X 0,Y 594.295,Z 543.853,A -85,B 0,C 180,E1 -1164.233,E2 -1164.233} C_VEL
LIN {X 0,Y 594.24,Z 548.94,A -85,B 0,C 180,E1 -1165.253,E2 -1165.253} C_VEL
LIN {X 0,Y 594.287,Z 552.88,A -85,B 0,C 180,E1 -1166.272,E2 -1166.272} C_VEL
LIN {X 0,Y 594.225,Z 555.791,A -85,B 0,C 180,E1 -1167.29,E2 -1167.29} C_VEL
LIN {X 0,Y 594.239,Z 557.201,A -85,B 0,C 180,E1 -1167.968,E2 -1167.968} C_VEL
LIN {X 0,Y 594.246,Z 558.186,A -85,B 0,C 180,E1 -1168.646,E2 -1168.646} C_VEL
LIN {X 0,Y 594.23,Z 559,A -85,B 0,C 180,E1 -1170.001,E2 -1170.001} C_VEL
LIN {X 0,Y 594.247,Z 558.183,A -85,B 0,C 180,E1 -1171.357,E2 -1171.357} C_VEL
LIN {X 0,Y 594.239,Z 557.197,A -85,B 0,C 180,E1 -1172.034,E2 -1172.034} C_VEL
LIN {X 0,Y 594.225,Z 555.785,A -85,B 0,C 180,E1 -1172.713,E2 -1172.713} C_VEL
LIN {X 0,Y 594.288,Z 552.871,A -85,B 0,C 180,E1 -1173.73,E2 -1173.73} C_VEL
LIN {X 0,Y 594.24,Z 548.927,A -85,B 0,C 180,E1 -1174.75,E2 -1174.75} C_VEL
LIN {X 0,Y 594.296,Z 543.837,A -85,B 0,C 180,E1 -1175.77,E2 -1175.77} C_VEL
LIN {X 0,Y 594.312,Z 537.444,A -85,B 0,C 180,E1 -1176.792,E2 -1176.792} C_VEL
LIN {X 0,Y 594.341,Z 529.407,A -85,B 0,C 180,E1 -1177.816,E2 -1177.816} C_VEL
LIN {X 0,Y 594.377,Z 519.532,A -85,B 0,C 180,E1 -1178.843,E2 -1178.843} C_VEL
LIN {X 0,Y 594.447,Z 509.012,A -85,B 0,C 180,E1 -1179.7,E2 -1179.7} C_VEL
LIN {X 0,Y 594.477,Z 498.753,A -85,B 0,C 180,E1 -1180.387,E2 -1180.387} C_VEL
LIN {X 0,Y 594.559,Z 487.605,A -85,B 0,C 180,E1 -1180.976,E2 -1180.976} C_VEL
LIN {X 0,Y 594.57,Z 475.631,A -85,B 0,C 180,E1 -1181.465,E2 -1181.465} C_VEL
LIN {X 0,Y 594.615,Z 463.256,A -85,B 0,C 180,E1 -1181.829,E2 -1181.829} C_VEL
LIN {X 0,Y 594.658,Z 449.071,A -85,B 0,C 180,E1 -1182.088,E2 -1182.088} C_VEL
LIN {X 0,Y 594.592,Z 346.356,A -85,B 0,C 180,E1 -1183.335,E2 -1183.335} C_VEL
LIN {X 0,Y 594.479,Z 345.287,A -85,B 0,C 180,E1 -1183.372,E2 -1183.372} C_VEL
LIN {X 0,Y 594.588,Z 320.972,A -85,B 0,C 180,E1 -1186.127,E2 -1186.127} C_VEL
LIN {X 0,Y 594.73,Z 295.72,A -85,B 0,C 180,E1 -1189.027,E2 -1189.027} C_VEL
LIN {X 0,Y 594.828,Z 271.57,A -85,B 0,C 180,E1 -1191.849,E2 -1191.849} C_VEL
LIN {X 0,Y 594.476,Z 267.304,A -85,B 0,C 180,E1 -1192.368,E2 -1192.368} C_VEL
LIN {X 0,Y 594.307,Z 266.456,A -85,B 0,C 180,E1 -1192.515,E2 -1192.515} C_VEL
LIN {X 0,Y 594.344,Z 266.455,A -85,B 0,C 180,E1 -1195.193,E2 -1195.193} C_VEL
LIN {X 0,Y 594.333,Z 266.455,A -85,B 0,C 180,E1 -1197.517,E2 -1197.517} C_VEL
LIN {X 0,Y 594.353,Z 266.444,A -85,B 0,C 180,E1 -1200.323,E2 -1200.323} C_VEL
LIN {X 0,Y 594.361,Z 266.445,A -85,B 0,C 180,E1 -1202.949,E2 -1202.949} C_VEL
LIN {X 0,Y 594.339,Z 266.453,A -85,B 0,C 180,E1 -1205.407,E2 -1205.407} C_VEL
LIN {X 0,Y 594.376,Z 266.447,A -85,B 0,C 180,E1 -1207.939,E2 -1207.939} C_VEL
LIN {X 0,Y 594.364,Z 266.442,A -85,B 0,C 180,E1 -1210.821,E2 -1210.821} C_VEL
LIN {X 0,Y 594.366,Z 266.444,A -85,B 0,C 180,E1 -1213.296,E2 -1213.296} C_VEL
LIN {X 0,Y 594.363,Z 266.448,A -85,B 0,C 180,E1 -1216.157,E2 -1216.157} C_VEL
LIN {X 0,Y 594.373,Z 266.441,A -85,B 0,C 180,E1 -1219.174,E2 -1219.174} C_VEL
LIN {X 0,Y 594.371,Z 266.452,A -85,B 0,C 180,E1 -1222.059,E2 -1222.059} C_VEL
LIN {X 0,Y 594.368,Z 266.443,A -85,B 0,C 180,E1 -1224.669,E2 -1224.669} C_VEL
LIN {X 0,Y 594.358,Z 266.442,A -85,B 0,C 180,E1 -1227.085,E2 -1227.085} C_VEL
LIN {X 0,Y 594.372,Z 266.442,A -85,B 0,C 180,E1 -1229.667,E2 -1229.667} C_VEL
LIN {X 0,Y 594.373,Z 266.442,A -85,B 0,C 180,E1 -1231.773,E2 -1231.773} C_VEL
LIN {X 0,Y 594.372,Z 266.445,A -85,B 0,C 180,E1 -1234.056,E2 -1234.056} C_VEL
LIN {X 0,Y 594.376,Z 266.448,A -85,B 0,C 180,E1 -1236.296,E2 -1236.296} C_VEL
LIN {X 0,Y 594.376,Z 266.442,A -85,B 0,C 180,E1 -1239.224,E2 -1239.224} C_VEL
LIN {X 0,Y 594.37,Z 266.443,A -85,B 0,C 180,E1 -1242.096,E2 -1242.096} C_VEL
LIN {X 0,Y 594.355,Z 266.451,A -85,B 0,C 180,E1 -1244.922,E2 -1244.922} C_VEL
LIN {X 0,Y 594.365,Z 266.442,A -85,B 0,C 180,E1 -1247.712,E2 -1247.712} C_VEL
LIN {X 0,Y 594.364,Z 266.442,A -85,B 0,C 180,E1 -1249.784,E2 -1249.784} C_VEL
LIN {X 0,Y 594.39,Z 266.443,A -85,B 0,C 180,E1 -1252.527,E2 -1252.527} C_VEL
LIN {X 0,Y 594.365,Z 266.45,A -85,B 0,C 180,E1 -1255.253,E2 -1255.253} C_VEL
LIN {X 0,Y 594.346,Z 266.449,A -85,B 0,C 180,E1 -1258.137,E2 -1258.137} C_VEL
LIN {X 0,Y 594.474,Z 267.177,A -85,B 0,C 180,E1 -1258.307,E2 -1258.307} C_VEL
LIN {X 0,Y 594.524,Z 277.652,A -85,B 0,C 180,E1 -1260,E2 -1260} C_VEL
LIN {X 0,Y 594.525,Z 293.594,A -85,B 0,C 180,E1 -1262.541,E2 -1262.541} C_VEL
LIN {X 0,Y 594.411,Z 313.089,A -85,B 0,C 180,E1 -1265.598,E2 -1265.598} C_VEL
LIN {X 0,Y 594.354,Z 330.723,A -85,B 0,C 180,E1 -1268.329,E2 -1268.329} C_VEL
LIN {X 0,Y 594.36,Z 338.664,A -85,B 0,C 180,E1 -1269.551,E2 -1269.551} C_VEL
LIN {X 0,Y 594.54,Z 353.425,A -85,B 0,C 180,E1 -1269.741,E2 -1269.741} C_VEL
LIN {X 0,Y 594.536,Z 392.413,A -85,B 0,C 180,E1 -1270.209,E2 -1270.209} C_VEL
LIN {X 0,Y 593.87,Z 398.271,A -85,B 0,C 180,E1 -1270.264,E2 -1270.264} C_VEL
LIN {X 0,Y 588.311,Z 416.245,A -85,B 0,C 180,E1 -1270.405,E2 -1270.405} C_VEL
LIN {X 0,Y 587.473,Z 422.015,A -85,B 0,C 180,E1 -1270.514,E2 -1270.514} C_VEL
LIN {X 0,Y 587.458,Z 422.92,A -85,B 0,C 180,E1 -1270.538,E2 -1270.538} C_VEL
LIN {X 0,Y 587.422,Z 432.374,A -85,B 0,C 180,E1 -1270.818,E2 -1270.818} C_VEL
LIN {X 0,Y 587.429,Z 440.567,A -85,B 0,C 180,E1 -1271.145,E2 -1271.145} C_VEL
LIN {X 0,Y 587.403,Z 448.462,A -85,B 0,C 180,E1 -1271.544,E2 -1271.544} C_VEL
LIN {X 0,Y 587.315,Z 457.105,A -85,B 0,C 180,E1 -1272.088,E2 -1272.088} C_VEL
LIN {X 0,Y 587.282,Z 464.985,A -85,B 0,C 180,E1 -1272.703,E2 -1272.703} C_VEL
LIN {X 0,Y 587.266,Z 473.231,A -85,B 0,C 180,E1 -1273.496,E2 -1273.496} C_VEL
LIN {X 0,Y 587.214,Z 480.014,A -85,B 0,C 180,E1 -1274.317,E2 -1274.317} C_VEL
LIN {X 0,Y 587.182,Z 486.145,A -85,B 0,C 180,E1 -1275.267,E2 -1275.267} C_VEL
LIN {X 0,Y 587.172,Z 491.44,A -85,B 0,C 180,E1 -1276.337,E2 -1276.337} C_VEL
LIN {X 0,Y 587.136,Z 495.294,A -85,B 0,C 180,E1 -1277.413,E2 -1277.413} C_VEL
LIN {X 0,Y 587.127,Z 497.022,A -85,B 0,C 180,E1 -1278.133,E2 -1278.133} C_VEL
LIN {X 0,Y 587.129,Z 498.372,A -85,B 0,C 180,E1 -1278.991,E2 -1278.991} C_VEL
LIN {X 0,Y 587.104,Z 498.815,A -85,B 0,C 180,E1 -1279.584,E2 -1279.584} C_VEL
LIN {X 0,Y 587.148,Z 498.904,A -85,B 0,C 180,E1 -1280.312,E2 -1280.312} C_VEL
LIN {X 0,Y 587.149,Z 498.445,A -85,B 0,C 180,E1 -1281.045,E2 -1281.045} C_VEL
LIN {X 0,Y 587.141,Z 497.403,A -85,B 0,C 180,E1 -1281.782,E2 -1281.782} C_VEL
LIN {X 0,Y 587.153,Z 494.764,A -85,B 0,C 180,E1 -1282.84,E2 -1282.84} C_VEL
LIN {X 0,Y 587.184,Z 491.945,A -85,B 0,C 180,E1 -1283.639,E2 -1283.639} C_VEL
LIN {X 0,Y 587.179,Z 487.649,A -85,B 0,C 180,E1 -1284.552,E2 -1284.552} C_VEL
LIN {X 0,Y 587.218,Z 483.02,A -85,B 0,C 180,E1 -1285.333,E2 -1285.333} C_VEL
LIN {X 0,Y 587.235,Z 476.886,A -85,B 0,C 180,E1 -1286.165,E2 -1286.165} C_VEL
LIN {X 0,Y 587.256,Z 470.64,A -85,B 0,C 180,E1 -1286.858,E2 -1286.858} C_VEL
LIN {X 0,Y 587.311,Z 462.942,A -85,B 0,C 180,E1 -1287.56,E2 -1287.56} C_VEL
LIN {X 0,Y 587.385,Z 452.67,A -85,B 0,C 180,E1 -1288.302,E2 -1288.302} C_VEL
LIN {X 0,Y 587.41,Z 444.379,A -85,B 0,C 180,E1 -1288.767,E2 -1288.767} C_VEL
LIN {X 0,Y 587.468,Z 435.414,A -85,B 0,C 180,E1 -1289.162,E2 -1289.162} C_VEL
LIN {X 0,Y 587.484,Z 425.546,A -85,B 0,C 180,E1 -1289.483,E2 -1289.483} C_VEL
LIN {X 0,Y 587.483,Z 416.075,A -85,B 0,C 180,E1 -1289.693,E2 -1289.693} C_VEL
LIN {X 0,Y 587.513,Z 340.539,A -85,B 0,C 180,E1 -1290.631,E2 -1290.631} C_VEL
LIN {X 0,Y 587.276,Z 338.58,A -85,B 0,C 180,E1 -1290.68,E2 -1290.68} C_VEL
LIN {X 0,Y 587.332,Z 319.866,A -85,B 0,C 180,E1 -1293.603,E2 -1293.603} C_VEL
LIN {X 0,Y 587.449,Z 302.728,A -85,B 0,C 180,E1 -1296.308,E2 -1296.308} C_VEL
LIN {X 0,Y 587.556,Z 286.07,A -85,B 0,C 180,E1 -1298.973,E2 -1298.973} C_VEL
LIN {X 0,Y 587.685,Z 269.996,A -85,B 0,C 180,E1 -1301.584,E2 -1301.584} C_VEL
LIN {X 0,Y 587.291,Z 267.328,A -85,B 0,C 180,E1 -1302.078,E2 -1302.078} C_VEL
LIN {X 0,Y 587.29,Z 267.334,A -85,B 0,C 180,E1 -1305.09,E2 -1305.09} C_VEL
LIN {X 0,Y 587.34,Z 267.318,A -85,B 0,C 180,E1 -1307.93,E2 -1307.93} C_VEL
LIN {X 0,Y 587.303,Z 267.324,A -85,B 0,C 180,E1 -1311.063,E2 -1311.063} C_VEL
LIN {X 0,Y 587.308,Z 267.325,A -85,B 0,C 180,E1 -1313.299,E2 -1313.299} C_VEL
LIN {X 0,Y 587.337,Z 267.328,A -85,B 0,C 180,E1 -1315.781,E2 -1315.781} C_VEL
LIN {X 0,Y 587.326,Z 267.323,A -85,B 0,C 180,E1 -1318.232,E2 -1318.232} C_VEL
LIN {X 0,Y 587.296,Z 267.322,A -85,B 0,C 180,E1 -1320.877,E2 -1320.877} C_VEL
LIN {X 0,Y 587.306,Z 267.324,A -85,B 0,C 180,E1 -1323.831,E2 -1323.831} C_VEL
LIN {X 0,Y 587.29,Z 267.327,A -85,B 0,C 180,E1 -1326.741,E2 -1326.741} C_VEL
LIN {X 0,Y 587.302,Z 267.321,A -85,B 0,C 180,E1 -1329.695,E2 -1329.695} C_VEL
LIN {X 0,Y 587.275,Z 267.324,A -85,B 0,C 180,E1 -1331.872,E2 -1331.872} C_VEL
LIN {X 0,Y 587.293,Z 267.322,A -85,B 0,C 180,E1 -1334.024,E2 -1334.024} C_VEL
LIN {X 0,Y 587.297,Z 267.331,A -85,B 0,C 180,E1 -1336.858,E2 -1336.858} C_VEL
LIN {X 0,Y 587.299,Z 267.324,A -85,B 0,C 180,E1 -1339.659,E2 -1339.659} C_VEL
LIN {X 0,Y 587.303,Z 267.321,A -85,B 0,C 180,E1 -1342.435,E2 -1342.435} C_VEL
LIN {X 0,Y 587.352,Z 267.321,A -85,B 0,C 180,E1 -1345.194,E2 -1345.194} C_VEL
LIN {X 0,Y 587.359,Z 267.319,A -85,B 0,C 180,E1 -1347.942,E2 -1347.942} C_VEL
LIN {X 0,Y 587.382,Z 267.317,A -85,B 0,C 180,E1 -1349.999,E2 -1349.999} C_VEL
LIN {X 0,Y 587.336,Z 267.316,A -85,B 0,C 180,E1 -1352.742,E2 -1352.742} C_VEL
LIN {X 0,Y 587.319,Z 267.321,A -85,B 0,C 180,E1 -1355.491,E2 -1355.491} C_VEL
LIN {X 0,Y 587.319,Z 267.33,A -85,B 0,C 180,E1 -1358.254,E2 -1358.254} C_VEL
LIN {X 0,Y 587.33,Z 267.318,A -85,B 0,C 180,E1 -1361.122,E2 -1361.122} C_VEL
LIN {X 0,Y 587.322,Z 267.319,A -85,B 0,C 180,E1 -1363.844,E2 -1363.844} C_VEL
LIN {X 0,Y 587.345,Z 267.325,A -85,B 0,C 180,E1 -1366.811,E2 -1366.811} C_VEL
LIN {X 0,Y 587.289,Z 267.323,A -85,B 0,C 180,E1 -1369.573,E2 -1369.573} C_VEL
LIN {X 0,Y 587.294,Z 267.322,A -85,B 0,C 180,E1 -1371.772,E2 -1371.772} C_VEL
LIN {X 0,Y 587.289,Z 267.327,A -85,B 0,C 180,E1 -1374.757,E2 -1374.757} C_VEL
LIN {X 0,Y 587.298,Z 267.326,A -85,B 0,C 180,E1 -1377.682,E2 -1377.682} C_VEL
LIN {X 0,Y 587.295,Z 267.322,A -85,B 0,C 180,E1 -1380.167,E2 -1380.167} C_VEL
LIN {X 0,Y 587.306,Z 267.32,A -85,B 0,C 180,E1 -1382.576,E2 -1382.576} C_VEL
LIN {X 0,Y 587.293,Z 267.323,A -85,B 0,C 180,E1 -1385.052,E2 -1385.052} C_VEL
LIN {X 0,Y 587.318,Z 267.329,A -85,B 0,C 180,E1 -1387.835,E2 -1387.835} C_VEL
LIN {X 0,Y 587.289,Z 267.33,A -85,B 0,C 180,E1 -1390.25,E2 -1390.25} C_VEL
LIN {X 0,Y 587.29,Z 267.322,A -85,B 0,C 180,E1 -1393.001,E2 -1393.001} C_VEL
LIN {X 0,Y 587.287,Z 267.328,A -85,B 0,C 180,E1 -1396.046,E2 -1396.046} C_VEL
LIN {X 0,Y 587.324,Z 267.322,A -85,B 0,C 180,E1 -1398.918,E2 -1398.918} C_VEL
LIN {X 0,Y 587.282,Z 267.323,A -85,B 0,C 180,E1 -1401.516,E2 -1401.516} C_VEL
LIN {X 0,Y 587.299,Z 267.322,A -85,B 0,C 180,E1 -1404.1,E2 -1404.1} C_VEL
LIN {X 0,Y 587.289,Z 267.332,A -85,B 0,C 180,E1 -1406.885,E2 -1406.885} C_VEL
LIN {X 0,Y 587.293,Z 267.327,A -85,B 0,C 180,E1 -1409.485,E2 -1409.485} C_VEL
LIN {X 0,Y 587.3,Z 267.321,A -85,B 0,C 180,E1 -1412.179,E2 -1412.179} C_VEL
LIN {X 0,Y 587.28,Z 267.323,A -85,B 0,C 180,E1 -1414.48,E2 -1414.48} C_VEL
LIN {X 0,Y 587.32,Z 267.328,A -85,B 0,C 180,E1 -1417.485,E2 -1417.485} C_VEL
LIN {X 0,Y 587.29,Z 267.323,A -85,B 0,C 180,E1 -1420.423,E2 -1420.423} C_VEL
LIN {X 0,Y 587.296,Z 267.323,A -85,B 0,C 180,E1 -1423.309,E2 -1423.309} C_VEL
LIN {X 0,Y 587.326,Z 267.329,A -85,B 0,C 180,E1 -1426.153,E2 -1426.153} C_VEL
LIN {X 0,Y 587.271,Z 267.325,A -85,B 0,C 180,E1 -1428.961,E2 -1428.961} C_VEL
LIN {X 0,Y 587.31,Z 267.321,A -85,B 0,C 180,E1 -1431.744,E2 -1431.744} C_VEL
LIN {X 0,Y 587.342,Z 267.326,A -85,B 0,C 180,E1 -1434.507,E2 -1434.507} C_VEL
LIN {X 0,Y 587.319,Z 267.321,A -85,B 0,C 180,E1 -1437.256,E2 -1437.256} C_VEL
LIN {X 0,Y 587.306,Z 267.32,A -85,B 0,C 180,E1 -1440,E2 -1440} C_VEL
LIN {X 0,Y 587.324,Z 267.324,A -85,B 0,C 180,E1 -1442.743,E2 -1442.743} C_VEL
LIN {X 0,Y 587.34,Z 267.322,A -85,B 0,C 180,E1 -1445.493,E2 -1445.493} C_VEL
LIN {X 0,Y 587.305,Z 267.32,A -85,B 0,C 180,E1 -1448.256,E2 -1448.256} C_VEL
LIN {X 0,Y 587.279,Z 267.328,A -85,B 0,C 180,E1 -1451.135,E2 -1451.135} C_VEL
LIN {X 0,Y 587.329,Z 267.319,A -85,B 0,C 180,E1 -1454.274,E2 -1454.274} C_VEL
LIN {X 0,Y 587.299,Z 267.324,A -85,B 0,C 180,E1 -1457.407,E2 -1457.407} C_VEL
LIN {X 0,Y 587.278,Z 267.33,A -85,B 0,C 180,E1 -1460.306,E2 -1460.306} C_VEL
LIN {X 0,Y 587.308,Z 267.32,A -85,B 0,C 180,E1 -1463.259,E2 -1463.259} C_VEL
LIN {X 0,Y 587.303,Z 267.33,A -85,B 0,C 180,E1 -1466.28,E2 -1466.28} C_VEL
LIN {X 0,Y 587.301,Z 267.323,A -85,B 0,C 180,E1 -1469.138,E2 -1469.138} C_VEL
LIN {X 0,Y 587.288,Z 267.322,A -85,B 0,C 180,E1 -1471.839,E2 -1471.839} C_VEL
LIN {X 0,Y 587.304,Z 267.323,A -85,B 0,C 180,E1 -1474.352,E2 -1474.352} C_VEL
LIN {X 0,Y 587.303,Z 267.327,A -85,B 0,C 180,E1 -1476.75,E2 -1476.75} C_VEL
LIN {X 0,Y 587.294,Z 267.329,A -85,B 0,C 180,E1 -1479.363,E2 -1479.363} C_VEL
LIN {X 0,Y 587.262,Z 267.326,A -85,B 0,C 180,E1 -1482.108,E2 -1482.108} C_VEL
LIN {X 0,Y 587.258,Z 267.328,A -85,B 0,C 180,E1 -1484.917,E2 -1484.917} C_VEL
LIN {X 0,Y 587.316,Z 267.325,A -85,B 0,C 180,E1 -1487.931,E2 -1487.931} C_VEL
LIN {X 0,Y 587.285,Z 267.323,A -85,B 0,C 180,E1 -1490.642,E2 -1490.642} C_VEL
LIN {X 0,Y 587.283,Z 267.324,A -85,B 0,C 180,E1 -1493.301,E2 -1493.301} C_VEL
LIN {X 0,Y 587.317,Z 267.325,A -85,B 0,C 180,E1 -1495.783,E2 -1495.783} C_VEL
LIN {X 0,Y 587.305,Z 267.333,A -85,B 0,C 180,E1 -1498.234,E2 -1498.234} C_VEL
LIN {X 0,Y 587.273,Z 267.328,A -85,B 0,C 180,E1 -1500.879,E2 -1500.879} C_VEL
LIN {X 0,Y 587.281,Z 267.325,A -85,B 0,C 180,E1 -1503.834,E2 -1503.834} C_VEL
LIN {X 0,Y 587.266,Z 267.336,A -85,B 0,C 180,E1 -1506.743,E2 -1506.743} C_VEL
LIN {X 0,Y 587.274,Z 267.446,A -85,B 0,C 180,E1 -1507.36,E2 -1507.36} C_VEL
LIN {X 0,Y 587.956,Z 271.595,A -85,B 0,C 180,E1 -1507.885,E2 -1507.885} C_VEL
LIN {X 0,Y 587.832,Z 294.298,A -85,B 0,C 180,E1 -1510.574,E2 -1510.574} C_VEL
LIN {X 0,Y 587.642,Z 317.909,A -85,B 0,C 180,E1 -1513.323,E2 -1513.323} C_VEL
LIN {X 0,Y 587.512,Z 342.61,A -85,B 0,C 180,E1 -1516.161,E2 -1516.161} C_VEL
LIN {X 0,Y 587.499,Z 345.581,A -85,B 0,C 180,E1 -1516.491,E2 -1516.491} C_VEL
LIN {X 0,Y 587.866,Z 350.946,A -85,B 0,C 180,E1 -1516.566,E2 -1516.566} C_VEL
LIN {X 0,Y 587.727,Z 454.885,A -85,B 0,C 180,E1 -1517.858,E2 -1517.858} C_VEL
LIN {X 0,Y 587.657,Z 466.713,A -85,B 0,C 180,E1 -1518.119,E2 -1518.119} C_VEL
LIN {X 0,Y 587.593,Z 479.521,A -85,B 0,C 180,E1 -1518.541,E2 -1518.541} C_VEL
LIN {X 0,Y 587.547,Z 492.676,A -85,B 0,C 180,E1 -1519.143,E2 -1519.143} C_VEL
LIN {X 0,Y 587.411,Z 504.168,A -85,B 0,C 180,E1 -1519.838,E2 -1519.838} C_VEL
LIN {X 0,Y 587.377,Z 513.495,A -85,B 0,C 180,E1 -1520.533,E2 -1520.533} C_VEL
LIN {X 0,Y 587.331,Z 521.314,A -85,B 0,C 180,E1 -1521.227,E2 -1521.227} C_VEL
LIN {X 0,Y 587.282,Z 529.43,A -85,B 0,C 180,E1 -1522.092,E2 -1522.092} C_VEL
LIN {X 0,Y 587.239,Z 536.252,A -85,B 0,C 180,E1 -1522.956,E2 -1522.956} C_VEL
LIN {X 0,Y 587.207,Z 541.879,A -85,B 0,C 180,E1 -1523.818,E2 -1523.818} C_VEL
LIN {X 0,Y 587.166,Z 547.374,A -85,B 0,C 180,E1 -1524.852,E2 -1524.852} C_VEL
LIN {X 0,Y 587.18,Z 551.682,A -85,B 0,C 180,E1 -1525.884,E2 -1525.884} C_VEL
LIN {X 0,Y 587.192,Z 553.962,A -85,B 0,C 180,E1 -1526.571,E2 -1526.571} C_VEL
LIN {X 0,Y 587.138,Z 557.2,A -85,B 0,C 180,E1 -1527.944,E2 -1527.944} C_VEL
LIN {X 0,Y 587.146,Z 558.187,A -85,B 0,C 180,E1 -1528.63,E2 -1528.63} C_VEL
LIN {X 0,Y 587.131,Z 559,A -85,B 0,C 180,E1 -1530.001,E2 -1530.001} C_VEL
LIN {X 0,Y 587.146,Z 558.184,A -85,B 0,C 180,E1 -1531.373,E2 -1531.373} C_VEL
LIN {X 0,Y 587.138,Z 557.197,A -85,B 0,C 180,E1 -1532.059,E2 -1532.059} C_VEL
LIN {X 0,Y 587.192,Z 553.954,A -85,B 0,C 180,E1 -1533.432,E2 -1533.432} C_VEL
LIN {X 0,Y 587.187,Z 550.367,A -85,B 0,C 180,E1 -1534.463,E2 -1534.463} C_VEL
LIN {X 0,Y 587.209,Z 545.674,A -85,B 0,C 180,E1 -1535.495,E2 -1535.495} C_VEL
LIN {X 0,Y 587.242,Z 539.108,A -85,B 0,C 180,E1 -1536.625,E2 -1536.625} C_VEL
LIN {X 0,Y 587.267,Z 532.25,A -85,B 0,C 180,E1 -1537.565,E2 -1537.565} C_VEL
LIN {X 0,Y 587.293,Z 526.386,A -85,B 0,C 180,E1 -1538.257,E2 -1538.257} C_VEL
LIN {X 0,Y 587.373,Z 517.525,A -85,B 0,C 180,E1 -1539.123,E2 -1539.123} C_VEL
LIN {X 0,Y 587.431,Z 509.015,A -85,B 0,C 180,E1 -1539.816,E2 -1539.816} C_VEL
LIN {X 0,Y 587.494,Z 498.745,A -85,B 0,C 180,E1 -1540.512,E2 -1540.512} C_VEL
LIN {X 0,Y 587.579,Z 488.491,A -85,B 0,C 180,E1 -1541.066,E2 -1541.066} C_VEL
LIN {X 0,Y 587.596,Z 477.11,A -85,B 0,C 180,E1 -1541.549,E2 -1541.549} C_VEL
LIN {X 0,Y 587.665,Z 464.937,A -85,B 0,C 180,E1 -1541.927,E2 -1541.927} C_VEL
LIN {X 0,Y 587.717,Z 453.418,A -85,B 0,C 180,E1 -1542.167,E2 -1542.167} C_VEL
LIN {X 0,Y 587.701,Z 347.138,A -85,B 0,C 180,E1 -1543.485,E2 -1543.485} C_VEL
LIN {X 0,Y 587.494,Z 345.287,A -85,B 0,C 180,E1 -1543.534,E2 -1543.534} C_VEL
LIN {X 0,Y 587.63,Z 319.428,A -85,B 0,C 180,E1 -1546.502,E2 -1546.502} C_VEL
LIN {X 0,Y 587.837,Z 294.279,A -85,B 0,C 180,E1 -1549.428,E2 -1549.428} C_VEL
LIN {X 0,Y 587.952,Z 271.57,A -85,B 0,C 180,E1 -1552.118,E2 -1552.118} C_VEL
LIN {X 0,Y 587.27,Z 267.334,A -85,B 0,C 180,E1 -1552.686,E2 -1552.686} C_VEL
LIN {X 0,Y 587.3,Z 267.33,A -85,B 0,C 180,E1 -1555.517,E2 -1555.517} C_VEL
LIN {X 0,Y 587.278,Z 267.329,A -85,B 0,C 180,E1 -1557.82,E2 -1557.82} C_VEL
LIN {X 0,Y 587.305,Z 267.322,A -85,B 0,C 180,E1 -1560.505,E2 -1560.505} C_VEL
LIN {X 0,Y 587.323,Z 267.328,A -85,B 0,C 180,E1 -1563.395,E2 -1563.395} C_VEL
LIN {X 0,Y 587.289,Z 267.329,A -85,B 0,C 180,E1 -1565.898,E2 -1565.898} C_VEL
LIN {X 0,Y 587.317,Z 267.32,A -85,B 0,C 180,E1 -1568.478,E2 -1568.478} C_VEL
LIN {X 0,Y 587.32,Z 267.322,A -85,B 0,C 180,E1 -1571.155,E2 -1571.155} C_VEL
LIN {X 0,Y 587.315,Z 267.329,A -85,B 0,C 180,E1 -1573.948,E2 -1573.948} C_VEL
LIN {X 0,Y 587.301,Z 267.322,A -85,B 0,C 180,E1 -1576.993,E2 -1576.993} C_VEL
LIN {X 0,Y 587.31,Z 267.327,A -85,B 0,C 180,E1 -1579.746,E2 -1579.746} C_VEL
LIN {X 0,Y 587.327,Z 267.324,A -85,B 0,C 180,E1 -1582.391,E2 -1582.391} C_VEL
LIN {X 0,Y 587.333,Z 267.317,A -85,B 0,C 180,E1 -1584.945,E2 -1584.945} C_VEL
LIN {X 0,Y 587.32,Z 267.319,A -85,B 0,C 180,E1 -1587.42,E2 -1587.42} C_VEL
LIN {X 0,Y 587.321,Z 267.322,A -85,B 0,C 180,E1 -1589.83,E2 -1589.83} C_VEL
LIN {X 0,Y 587.321,Z 267.329,A -85,B 0,C 180,E1 -1592.305,E2 -1592.305} C_VEL
LIN {X 0,Y 587.326,Z 267.329,A -85,B 0,C 180,E1 -1594.483,E2 -1594.483} C_VEL
LIN {X 0,Y 587.343,Z 267.316,A -85,B 0,C 180,E1 -1597.487,E2 -1597.487} C_VEL
LIN {X 0,Y 587.321,Z 267.327,A -85,B 0,C 180,E1 -1600.425,E2 -1600.425} C_VEL
LIN {X 0,Y 587.319,Z 267.321,A -85,B 0,C 180,E1 -1603.311,E2 -1603.311} C_VEL
LIN {X 0,Y 587.35,Z 267.317,A -85,B 0,C 180,E1 -1606.154,E2 -1606.154} C_VEL
LIN {X 0,Y 587.372,Z 267.323,A -85,B 0,C 180,E1 -1608.963,E2 -1608.963} C_VEL
LIN {X 0,Y 587.332,Z 267.319,A -85,B 0,C 180,E1 -1611.745,E2 -1611.745} C_VEL
LIN {X 0,Y 587.341,Z 267.32,A -85,B 0,C 180,E1 -1614.507,E2 -1614.507} C_VEL
LIN {X 0,Y 587.347,Z 267.326,A -85,B 0,C 180,E1 -1617.257,E2 -1617.257} C_VEL
LIN {X 0,Y 587.317,Z 267.442,A -85,B 0,C 180,E1 -1618.072,E2 -1618.072} C_VEL
LIN {X 0,Y 587.67,Z 271.801,A -85,B 0,C 180,E1 -1618.801,E2 -1618.801} C_VEL
LIN {X 0,Y 587.504,Z 288.724,A -85,B 0,C 180,E1 -1621.543,E2 -1621.543} C_VEL
LIN {X 0,Y 587.437,Z 303.757,A -85,B 0,C 180,E1 -1623.945,E2 -1623.945} C_VEL
LIN {X 0,Y 587.31,Z 317.934,A -85,B 0,C 180,E1 -1626.183,E2 -1626.183} C_VEL
LIN {X 0,Y 587.288,Z 333.398,A -85,B 0,C 180,E1 -1628.603,E2 -1628.603} C_VEL
LIN {X 0,Y 587.318,Z 338.689,A -85,B 0,C 180,E1 -1629.427,E2 -1629.427} C_VEL
LIN {X 0,Y 587.598,Z 349.882,A -85,B 0,C 180,E1 -1629.575,E2 -1629.575} C_VEL
LIN {X 0,Y 587.518,Z 416.333,A -85,B 0,C 180,E1 -1630.402,E2 -1630.402} C_VEL
LIN {X 0,Y 587.458,Z 422.92,A -85,B 0,C 180,E1 -1630.538,E2 -1630.538} C_VEL
LIN {X 0,Y 586.321,Z 430.661,A -85,B 0,C 180,E1 -1630.739,E2 -1630.739} C_VEL
LIN {X 0,Y 583.927,Z 438.079,A -85,B 0,C 180,E1 -1630.976,E2 -1630.976} C_VEL
LIN {X 0,Y 581.025,Z 446.616,A -85,B 0,C 180,E1 -1631.342,E2 -1631.342} C_VEL
LIN {X 0,Y 580.336,Z 451.479,A -85,B 0,C 180,E1 -1631.617,E2 -1631.617} C_VEL
LIN {X 0,Y 580.268,Z 461.633,A -85,B 0,C 180,E1 -1632.326,E2 -1632.326} C_VEL
LIN {X 0,Y 580.22,Z 468.696,A -85,B 0,C 180,E1 -1632.949,E2 -1632.949} C_VEL
LIN {X 0,Y 580.188,Z 475.36,A -85,B 0,C 180,E1 -1633.663,E2 -1633.663} C_VEL
LIN {X 0,Y 580.138,Z 482.303,A -85,B 0,C 180,E1 -1634.586,E2 -1634.586} C_VEL
LIN {X 0,Y 580.094,Z 487.518,A -85,B 0,C 180,E1 -1635.459,E2 -1635.459} C_VEL
LIN {X 0,Y 580.079,Z 492.399,A -85,B 0,C 180,E1 -1636.514,E2 -1636.514} C_VEL
LIN {X 0,Y 580.041,Z 495.92,A -85,B 0,C 180,E1 -1637.633,E2 -1637.633} C_VEL
LIN {X 0,Y 580.028,Z 497.529,A -85,B 0,C 180,E1 -1638.363,E2 -1638.363} C_VEL
LIN {X 0,Y 580.024,Z 498.529,A -85,B 0,C 180,E1 -1639.096,E2 -1639.096} C_VEL
LIN {X 0,Y 580.036,Z 498.929,A -85,B 0,C 180,E1 -1639.832,E2 -1639.832} C_VEL
LIN {X 0,Y 580.045,Z 498.373,A -85,B 0,C 180,E1 -1641.111,E2 -1641.111} C_VEL
LIN {X 0,Y 580.037,Z 496.832,A -85,B 0,C 180,E1 -1642.062,E2 -1642.062} C_VEL
LIN {X 0,Y 580.071,Z 494.459,A -85,B 0,C 180,E1 -1642.967,E2 -1642.967} C_VEL
LIN {X 0,Y 580.089,Z 492.435,A -85,B 0,C 180,E1 -1643.567,E2 -1643.567} C_VEL
LIN {X 0,Y 580.099,Z 489.134,A -85,B 0,C 180,E1 -1644.326,E2 -1644.326} C_VEL
LIN {X 0,Y 580.121,Z 483.806,A -85,B 0,C 180,E1 -1645.281,E2 -1645.281} C_VEL
LIN {X 0,Y 580.165,Z 478.123,A -85,B 0,C 180,E1 -1646.087,E2 -1646.087} C_VEL
LIN {X 0,Y 580.182,Z 471.793,A -85,B 0,C 180,E1 -1646.823,E2 -1646.823} C_VEL
LIN {X 0,Y 580.238,Z 465.818,A -85,B 0,C 180,E1 -1647.405,E2 -1647.405} C_VEL
LIN {X 0,Y 580.276,Z 458.879,A -85,B 0,C 180,E1 -1647.972,E2 -1647.972} C_VEL
LIN {X 0,Y 580.35,Z 449.705,A -85,B 0,C 180,E1 -1648.578,E2 -1648.578} C_VEL
LIN {X 0,Y 580.401,Z 440.987,A -85,B 0,C 180,E1 -1649.033,E2 -1649.033} C_VEL
LIN {X 0,Y 580.479,Z 431.395,A -85,B 0,C 180,E1 -1649.419,E2 -1649.419} C_VEL
LIN {X 0,Y 580.502,Z 419.852,A -85,B 0,C 180,E1 -1649.744,E2 -1649.744} C_VEL
LIN {X 0,Y 580.554,Z 403.534,A -85,B 0,C 180,E1 -1649.983,E2 -1649.983} C_VEL
LIN {X 0,Y 580.48,Z 340.811,A -85,B 0,C 180,E1 -1650.757,E2 -1650.757} C_VEL
LIN {X 0,Y 580.231,Z 338.689,A -85,B 0,C 180,E1 -1650.794,E2 -1650.794} C_VEL
LIN {X 0,Y 580.307,Z 321.199,A -85,B 0,C 180,E1 -1653.558,E2 -1653.558} C_VEL
LIN {X 0,Y 580.437,Z 304.519,A -85,B 0,C 180,E1 -1656.222,E2 -1656.222} C_VEL
LIN {X 0,Y 580.552,Z 288.64,A -85,B 0,C 180,E1 -1658.791,E2 -1658.791} C_VEL
LIN {X 0,Y 580.746,Z 272.127,A -85,B 0,C 180,E1 -1661.501,E2 -1661.501} C_VEL
LIN {X 0,Y 580.275,Z 268.204,A -85,B 0,C 180,E1 -1662.162,E2 -1662.162} C_VEL
LIN {X 0,Y 580.238,Z 268.205,A -85,B 0,C 180,E1 -1664.629,E2 -1664.629} C_VEL
LIN {X 0,Y 580.275,Z 268.202,A -85,B 0,C 180,E1 -1667.63,E2 -1667.63} C_VEL
LIN {X 0,Y 580.268,Z 268.198,A -85,B 0,C 180,E1 -1670.068,E2 -1670.068} C_VEL
LIN {X 0,Y 580.263,Z 268.2,A -85,B 0,C 180,E1 -1673.071,E2 -1673.071} C_VEL
LIN {X 0,Y 580.296,Z 268.198,A -85,B 0,C 180,E1 -1676.146,E2 -1676.146} C_VEL
LIN {X 0,Y 580.26,Z 268.199,A -85,B 0,C 180,E1 -1678.615,E2 -1678.615} C_VEL
LIN {X 0,Y 580.242,Z 268.2,A -85,B 0,C 180,E1 -1681.023,E2 -1681.023} C_VEL
LIN {X 0,Y 580.26,Z 268.2,A -85,B 0,C 180,E1 -1683.673,E2 -1683.673} C_VEL
LIN {X 0,Y 580.244,Z 268.211,A -85,B 0,C 180,E1 -1686.442,E2 -1686.442} C_VEL
LIN {X 0,Y 580.251,Z 268.199,A -85,B 0,C 180,E1 -1689.437,E2 -1689.437} C_VEL
LIN {X 0,Y 580.237,Z 268.201,A -85,B 0,C 180,E1 -1691.644,E2 -1691.644} C_VEL
LIN {X 0,Y 580.248,Z 268.199,A -85,B 0,C 180,E1 -1693.825,E2 -1693.825} C_VEL
LIN {X 0,Y 580.279,Z 268.195,A -85,B 0,C 180,E1 -1695.982,E2 -1695.982} C_VEL
LIN {X 0,Y 580.311,Z 268.198,A -85,B 0,C 180,E1 -1698.827,E2 -1698.827} C_VEL
LIN {X 0,Y 580.291,Z 268.198,A -85,B 0,C 180,E1 -1701.643,E2 -1701.643} C_VEL
LIN {X 0,Y 580.286,Z 268.194,A -85,B 0,C 180,E1 -1704.439,E2 -1704.439} C_VEL
LIN {X 0,Y 580.317,Z 268.196,A -85,B 0,C 180,E1 -1707.222,E2 -1707.222} C_VEL
LIN {X 0,Y 580.35,Z 268.193,A -85,B 0,C 180,E1 -1709.999,E2 -1709.999} C_VEL
LIN {X 0,Y 580.303,Z 268.192,A -85,B 0,C 180,E1 -1712.775,E2 -1712.775} C_VEL
LIN {X 0,Y 580.289,Z 268.197,A -85,B 0,C 180,E1 -1715.558,E2 -1715.558} C_VEL
LIN {X 0,Y 580.291,Z 268.203,A -85,B 0,C 180,E1 -1718.354,E2 -1718.354} C_VEL
LIN {X 0,Y 580.301,Z 268.193,A -85,B 0,C 180,E1 -1721.188,E2 -1721.188} C_VEL
LIN {X 0,Y 580.286,Z 268.197,A -85,B 0,C 180,E1 -1724.015,E2 -1724.015} C_VEL
LIN {X 0,Y 580.309,Z 268.199,A -85,B 0,C 180,E1 -1726.911,E2 -1726.911} C_VEL
LIN {X 0,Y 580.265,Z 268.197,A -85,B 0,C 180,E1 -1729.82,E2 -1729.82} C_VEL
LIN {X 0,Y 580.238,Z 268.2,A -85,B 0,C 180,E1 -1732.05,E2 -1732.05} C_VEL
LIN {X 0,Y 580.268,Z 268.207,A -85,B 0,C 180,E1 -1735.077,E2 -1735.077} C_VEL
LIN {X 0,Y 580.259,Z 268.198,A -85,B 0,C 180,E1 -1738.183,E2 -1738.183} C_VEL
LIN {X 0,Y 580.249,Z 268.2,A -85,B 0,C 180,E1 -1740.688,E2 -1740.688} C_VEL
LIN {X 0,Y 580.28,Z 268.201,A -85,B 0,C 180,E1 -1743.312,E2 -1743.312} C_VEL
LIN {X 0,Y 580.239,Z 268.212,A -85,B 0,C 180,E1 -1745.755,E2 -1745.755} C_VEL
LIN {X 0,Y 580.262,Z 268.205,A -85,B 0,C 180,E1 -1748.142,E2 -1748.142} C_VEL
LIN {X 0,Y 580.267,Z 268.197,A -85,B 0,C 180,E1 -1750.839,E2 -1750.839} C_VEL
LIN {X 0,Y 580.238,Z 268.203,A -85,B 0,C 180,E1 -1753.654,E2 -1753.654} C_VEL
LIN {X 0,Y 580.238,Z 268.208,A -85,B 0,C 180,E1 -1756.605,E2 -1756.605} C_VEL
LIN {X 0,Y 580.277,Z 268.198,A -85,B 0,C 180,E1 -1759.154,E2 -1759.154} C_VEL
LIN {X 0,Y 580.244,Z 268.2,A -85,B 0,C 180,E1 -1761.923,E2 -1761.923} C_VEL
LIN {X 0,Y 580.257,Z 268.202,A -85,B 0,C 180,E1 -1764.453,E2 -1764.453} C_VEL
LIN {X 0,Y 580.242,Z 268.212,A -85,B 0,C 180,E1 -1766.972,E2 -1766.972} C_VEL
LIN {X 0,Y 580.253,Z 268.205,A -85,B 0,C 180,E1 -1769.422,E2 -1769.422} C_VEL
LIN {X 0,Y 580.27,Z 268.197,A -85,B 0,C 180,E1 -1772.133,E2 -1772.133} C_VEL
LIN {X 0,Y 580.252,Z 268.201,A -85,B 0,C 180,E1 -1774.917,E2 -1774.917} C_VEL
LIN {X 0,Y 580.274,Z 268.201,A -85,B 0,C 180,E1 -1777.196,E2 -1777.196} C_VEL
LIN {X 0,Y 580.254,Z 268.203,A -85,B 0,C 180,E1 -1780.175,E2 -1780.175} C_VEL
LIN {X 0,Y 580.267,Z 268.197,A -85,B 0,C 180,E1 -1783.101,E2 -1783.101} C_VEL
LIN {X 0,Y 580.29,Z 268.204,A -85,B 0,C 180,E1 -1785.982,E2 -1785.982} C_VEL
LIN {X 0,Y 580.237,Z 268.203,A -85,B 0,C 180,E1 -1788.825,E2 -1788.825} C_VEL
LIN {X 0,Y 580.273,Z 268.197,A -85,B 0,C 180,E1 -1791.643,E2 -1791.643} C_VEL
LIN {X 0,Y 580.301,Z 268.202,A -85,B 0,C 180,E1 -1794.44,E2 -1794.44} C_VEL
LIN {X 0,Y 580.286,Z 268.198,A -85,B 0,C 180,E1 -1797.223,E2 -1797.223} C_VEL
LIN {X 0,Y 580.276,Z 268.196,A -85,B 0,C 180,E1 -1800,E2 -1800} C_VEL
LIN {X 0,Y 580.29,Z 268.2,A -85,B 0,C 180,E1 -1802.776,E2 -1802.776} C_VEL
LIN {X 0,Y 580.298,Z 268.198,A -85,B 0,C 180,E1 -1805.56,E2 -1805.56} C_VEL
LIN {X 0,Y 580.269,Z 268.197,A -85,B 0,C 180,E1 -1808.357,E2 -1808.357} C_VEL
LIN {X 0,Y 580.231,Z 268.207,A -85,B 0,C 180,E1 -1811.192,E2 -1811.192} C_VEL
LIN {X 0,Y 580.289,Z 268.2,A -85,B 0,C 180,E1 -1814.017,E2 -1814.017} C_VEL
LIN {X 0,Y 580.246,Z 268.199,A -85,B 0,C 180,E1 -1816.915,E2 -1816.915} C_VEL
LIN {X 0,Y 580.249,Z 268.207,A -85,B 0,C 180,E1 -1819.824,E2 -1819.824} C_VEL
LIN {X 0,Y 580.267,Z 268.199,A -85,B 0,C 180,E1 -1822.803,E2 -1822.803} C_VEL
LIN {X 0,Y 580.246,Z 268.2,A -85,B 0,C 180,E1 -1825.082,E2 -1825.082} C_VEL
LIN {X 0,Y 580.266,Z 268.199,A -85,B 0,C 180,E1 -1827.866,E2 -1827.866} C_VEL
LIN {X 0,Y 580.229,Z 268.213,A -85,B 0,C 180,E1 -1830.698,E2 -1830.698} C_VEL
LIN {X 0,Y 580.231,Z 268.204,A -85,B 0,C 180,E1 -1833.317,E2 -1833.317} C_VEL
LIN {X 0,Y 580.246,Z 268.2,A -85,B 0,C 180,E1 -1835.767,E2 -1835.767} C_VEL
LIN {X 0,Y 580.236,Z 268.201,A -85,B 0,C 180,E1 -1838.15,E2 -1838.15} C_VEL
LIN {X 0,Y 580.254,Z 268.203,A -85,B 0,C 180,E1 -1840.847,E2 -1840.847} C_VEL
LIN {X 0,Y 580.235,Z 268.207,A -85,B 0,C 180,E1 -1843.661,E2 -1843.661} C_VEL
LIN {X 0,Y 580.234,Z 268.201,A -85,B 0,C 180,E1 -1846.613,E2 -1846.613} C_VEL
LIN {X 0,Y 580.258,Z 268.2,A -85,B 0,C 180,E1 -1849.16,E2 -1849.16} C_VEL
LIN {X 0,Y 580.251,Z 268.21,A -85,B 0,C 180,E1 -1851.932,E2 -1851.932} C_VEL
LIN {X 0,Y 580.202,Z 268.209,A -85,B 0,C 180,E1 -1854.455,E2 -1854.455} C_VEL
LIN {X 0,Y 580.214,Z 268.204,A -85,B 0,C 180,E1 -1856.976,E2 -1856.976} C_VEL
LIN {X 0,Y 580.249,Z 268.199,A -85,B 0,C 180,E1 -1859.427,E2 -1859.427} C_VEL
LIN {X 0,Y 580.213,Z 268.211,A -85,B 0,C 180,E1 -1862.157,E2 -1862.157} C_VEL
LIN {X 0,Y 580.258,Z 268.206,A -85,B 0,C 180,E1 -1864.922,E2 -1864.922} C_VEL
LIN {X 0,Y 580.244,Z 268.269,A -85,B 0,C 180,E1 -1867.172,E2 -1867.172} C_VEL
LIN {X 0,Y 581.08,Z 273.139,A -85,B 0,C 180,E1 -1867.796,E2 -1867.796} C_VEL
LIN {X 0,Y 580.915,Z 295.77,A -85,B 0,C 180,E1 -1870.508,E2 -1870.508} C_VEL
LIN {X 0,Y 580.652,Z 320.997,A -85,B 0,C 180,E1 -1873.478,E2 -1873.478} C_VEL
LIN {X 0,Y 580.501,Z 345.581,A -85,B 0,C 180,E1 -1876.325,E2 -1876.325} C_VEL
LIN {X 0,Y 580.965,Z 350.946,A -85,B 0,C 180,E1 -1876.403,E2 -1876.403} C_VEL
LIN {X 0,Y 580.802,Z 454.819,A -85,B 0,C 180,E1 -1877.711,E2 -1877.711} C_VEL
LIN {X 0,Y 580.693,Z 466.669,A -85,B 0,C 180,E1 -1877.974,E2 -1877.974} C_VEL
LIN {X 0,Y 580.643,Z 478.738,A -85,B 0,C 180,E1 -1878.372,E2 -1878.372} C_VEL
LIN {X 0,Y 580.573,Z 490.98,A -85,B 0,C 180,E1 -1878.923,E2 -1878.923} C_VEL
LIN {X 0,Y 580.439,Z 502.934,A -85,B 0,C 180,E1 -1879.626,E2 -1879.626} C_VEL
LIN {X 0,Y 580.36,Z 513.493,A -85,B 0,C 180,E1 -1880.418,E2 -1880.418} C_VEL
LIN {X 0,Y 580.305,Z 521.313,A -85,B 0,C 180,E1 -1881.12,E2 -1881.12} C_VEL
LIN {X 0,Y 580.236,Z 529.431,A -85,B 0,C 180,E1 -1881.995,E2 -1881.995} C_VEL
LIN {X 0,Y 580.179,Z 536.253,A -85,B 0,C 180,E1 -1882.87,E2 -1882.87} C_VEL
LIN {X 0,Y 580.13,Z 541.879,A -85,B 0,C 180,E1 -1883.743,E2 -1883.743} C_VEL
LIN {X 0,Y 580.084,Z 547.375,A -85,B 0,C 180,E1 -1884.788,E2 -1884.788} C_VEL
LIN {X 0,Y 580.103,Z 551.682,A -85,B 0,C 180,E1 -1885.833,E2 -1885.833} C_VEL
LIN {X 0,Y 580.121,Z 553.962,A -85,B 0,C 180,E1 -1886.529,E2 -1886.529} C_VEL
LIN {X 0,Y 580.037,Z 557.199,A -85,B 0,C 180,E1 -1887.918,E2 -1887.918} C_VEL
LIN {X 0,Y 580.046,Z 558.187,A -85,B 0,C 180,E1 -1888.613,E2 -1888.613} C_VEL
LIN {X 0,Y 580.031,Z 559,A -85,B 0,C 180,E1 -1890.001,E2 -1890.001} C_VEL
LIN {X 0,Y 580.046,Z 558.185,A -85,B 0,C 180,E1 -1891.39,E2 -1891.39} C_VEL
LIN {X 0,Y 580.037,Z 557.196,A -85,B 0,C 180,E1 -1892.084,E2 -1892.084} C_VEL
LIN {X 0,Y 580.121,Z 553.955,A -85,B 0,C 180,E1 -1893.474,E2 -1893.474} C_VEL
LIN {X 0,Y 580.107,Z 550.367,A -85,B 0,C 180,E1 -1894.518,E2 -1894.518} C_VEL
LIN {X 0,Y 580.135,Z 545.674,A -85,B 0,C 180,E1 -1895.562,E2 -1895.562} C_VEL
LIN {X 0,Y 580.166,Z 539.634,A -85,B 0,C 180,E1 -1896.624,E2 -1896.624} C_VEL
LIN {X 0,Y 580.197,Z 533.667,A -85,B 0,C 180,E1 -1897.483,E2 -1897.483} C_VEL
LIN {X 0,Y 580.247,Z 526.385,A -85,B 0,C 180,E1 -1898.358,E2 -1898.358} C_VEL
LIN {X 0,Y 580.332,Z 517.527,A -85,B 0,C 180,E1 -1899.234,E2 -1899.234} C_VEL
LIN {X 0,Y 580.4,Z 509.019,A -85,B 0,C 180,E1 -1899.937,E2 -1899.937} C_VEL
LIN {X 0,Y 580.499,Z 498.724,A -85,B 0,C 180,E1 -1900.64,E2 -1900.64} C_VEL
LIN {X 0,Y 580.604,Z 489.165,A -85,B 0,C 180,E1 -1901.168,E2 -1901.168} C_VEL
LIN {X 0,Y 580.633,Z 478.058,A -85,B 0,C 180,E1 -1901.653,E2 -1901.653} C_VEL
LIN {X 0,Y 580.699,Z 466.557,A -85,B 0,C 180,E1 -1902.028,E2 -1902.028} C_VEL
LIN {X 0,Y 580.803,Z 454.649,A -85,B 0,C 180,E1 -1902.292,E2 -1902.292} C_VEL
LIN {X 0,Y 580.822,Z 347.92,A -85,B 0,C 180,E1 -1903.638,E2 -1903.638} C_VEL
LIN {X 0,Y 580.5,Z 345.287,A -85,B 0,C 180,E1 -1903.7,E2 -1903.7} C_VEL
LIN {X 0,Y 580.678,Z 319.428,A -85,B 0,C 180,E1 -1906.705,E2 -1906.705} C_VEL
LIN {X 0,Y 580.967,Z 291.639,A -85,B 0,C 180,E1 -1909.982,E2 -1909.982} C_VEL
LIN {X 0,Y 581.076,Z 273.114,A -85,B 0,C 180,E1 -1912.207,E2 -1912.207} C_VEL
LIN {X 0,Y 580.24,Z 268.211,A -85,B 0,C 180,E1 -1912.859,E2 -1912.859} C_VEL
LIN {X 0,Y 580.243,Z 268.204,A -85,B 0,C 180,E1 -1915.85,E2 -1915.85} C_VEL
LIN {X 0,Y 580.224,Z 268.205,A -85,B 0,C 180,E1 -1918.188,E2 -1918.188} C_VEL
LIN {X 0,Y 580.256,Z 268.201,A -85,B 0,C 180,E1 -1920.69,E2 -1920.69} C_VEL
LIN {X 0,Y 580.291,Z 268.203,A -85,B 0,C 180,E1 -1923.315,E2 -1923.315} C_VEL
LIN {X 0,Y 580.251,Z 268.208,A -85,B 0,C 180,E1 -1925.758,E2 -1925.758} C_VEL
LIN {X 0,Y 580.275,Z 268.201,A -85,B 0,C 180,E1 -1928.145,E2 -1928.145} C_VEL
LIN {X 0,Y 580.286,Z 268.196,A -85,B 0,C 180,E1 -1930.841,E2 -1930.841} C_VEL
LIN {X 0,Y 580.271,Z 268.206,A -85,B 0,C 180,E1 -1933.655,E2 -1933.655} C_VEL
LIN {X 0,Y 580.265,Z 268.199,A -85,B 0,C 180,E1 -1936.607,E2 -1936.607} C_VEL
LIN {X 0,Y 580.3,Z 268.194,A -85,B 0,C 180,E1 -1939.157,E2 -1939.157} C_VEL
LIN {X 0,Y 580.27,Z 268.206,A -85,B 0,C 180,E1 -1941.925,E2 -1941.925} C_VEL
LIN {X 0,Y 580.287,Z 268.2,A -85,B 0,C 180,E1 -1944.456,E2 -1944.456} C_VEL
LIN {X 0,Y 580.271,Z 268.197,A -85,B 0,C 180,E1 -1946.974,E2 -1946.974} C_VEL
LIN {X 0,Y 580.283,Z 268.195,A -85,B 0,C 180,E1 -1949.425,E2 -1949.425} C_VEL
LIN {X 0,Y 580.292,Z 268.201,A -85,B 0,C 180,E1 -1952.135,E2 -1952.135} C_VEL
LIN {X 0,Y 580.29,Z 268.198,A -85,B 0,C 180,E1 -1954.92,E2 -1954.92} C_VEL
LIN {X 0,Y 580.304,Z 268.195,A -85,B 0,C 180,E1 -1957.949,E2 -1957.949} C_VEL
LIN {X 0,Y 580.281,Z 268.202,A -85,B 0,C 180,E1 -1960.913,E2 -1960.913} C_VEL
LIN {X 0,Y 580.262,Z 268.199,A -85,B 0,C 180,E1 -1963.825,E2 -1963.825} C_VEL
LIN {X 0,Y 580.313,Z 268.193,A -85,B 0,C 180,E1 -1965.983,E2 -1965.983} C_VEL
LIN {X 0,Y 580.351,Z 268.199,A -85,B 0,C 180,E1 -1968.828,E2 -1968.828} C_VEL
LIN {X 0,Y 580.297,Z 268.196,A -85,B 0,C 180,E1 -1971.644,E2 -1971.644} C_VEL
LIN {X 0,Y 580.303,Z 268.197,A -85,B 0,C 180,E1 -1974.44,E2 -1974.44} C_VEL
LIN {X 0,Y 580.313,Z 268.203,A -85,B 0,C 180,E1 -1977.224,E2 -1977.224} C_VEL
LIN {X 0,Y 580.289,Z 268.327,A -85,B 0,C 180,E1 -1977.962,E2 -1977.962} C_VEL
LIN {X 0,Y 580.727,Z 273.321,A -85,B 0,C 180,E1 -1978.787,E2 -1978.787} C_VEL
LIN {X 0,Y 580.52,Z 290.254,A -85,B 0,C 180,E1 -1981.561,E2 -1981.561} C_VEL
LIN {X 0,Y 580.384,Z 306.387,A -85,B 0,C 180,E1 -1984.167,E2 -1984.167} C_VEL
LIN {X 0,Y 580.341,Z 323.864,A -85,B 0,C 180,E1 -1986.956,E2 -1986.956} C_VEL
LIN {X 0,Y 580.273,Z 338.716,A -85,B 0,C 180,E1 -1989.301,E2 -1989.301} C_VEL
LIN {X 0,Y 580.615,Z 348.251,A -85,B 0,C 180,E1 -1989.427,E2 -1989.427} C_VEL
LIN {X 0,Y 580.541,Z 415.092,A -85,B 0,C 180,E1 -1990.264,E2 -1990.264} C_VEL
LIN {X 0,Y 580.47,Z 424.494,A -85,B 0,C 180,E1 -1990.464,E2 -1990.464} C_VEL
LIN {X 0,Y 580.447,Z 434.129,A -85,B 0,C 180,E1 -1990.77,E2 -1990.77} C_VEL
LIN {X 0,Y 580.418,Z 443.412,A -85,B 0,C 180,E1 -1991.171,E2 -1991.171} C_VEL
LIN {X 0,Y 580.336,Z 451.479,A -85,B 0,C 180,E1 -1991.617,E2 -1991.617} C_VEL
LIN {X 0,Y 579.66,Z 456.473,A -85,B 0,C 180,E1 -1991.925,E2 -1991.925} C_VEL
LIN {X 0,Y 576.719,Z 464.192,A -85,B 0,C 180,E1 -1992.474,E2 -1992.474} C_VEL
LIN {X 0,Y 573.783,Z 471.205,A -85,B 0,C 180,E1 -1993.11,E2 -1993.11} C_VEL
LIN {X 0,Y 573.115,Z 475.088,A -85,B 0,C 180,E1 -1993.551,E2 -1993.551} C_VEL
LIN {X 0,Y 573.069,Z 481.231,A -85,B 0,C 180,E1 -1994.358,E2 -1994.358} C_VEL
LIN {X 0,Y 573.056,Z 484.924,A -85,B 0,C 180,E1 -1994.925,E2 -1994.925} C_VEL
LIN {X 0,Y 573.009,Z 488.864,A -85,B 0,C 180,E1 -1995.655,E2 -1995.655} C_VEL
LIN {X 0,Y 572.989,Z 492.049,A -85,B 0,C 180,E1 -1996.386,E2 -1996.386} C_VEL
LIN {X 0,Y 572.967,Z 494.572,A -85,B 0,C 180,E1 -1997.121,E2 -1997.121} C_VEL
LIN {X 0,Y 572.937,Z 496.507,A -85,B 0,C 180,E1 -1997.859,E2 -1997.859} C_VEL
LIN {X 0,Y 572.933,Z 498.626,A -85,B 0,C 180,E1 -1999.184,E2 -1999.184} C_VEL
LIN {X 0,Y 572.959,Z 498.996,A -85,B 0,C 180,E1 -2000.088,E2 -2000.088} C_VEL
LIN {X 0,Y 572.958,Z 498.238,A -85,B 0,C 180,E1 -2001.226,E2 -2001.226} C_VEL
LIN {X 0,Y 572.946,Z 496.233,A -85,B 0,C 180,E1 -2002.35,E2 -2002.35} C_VEL
LIN {X 0,Y 573,Z 494.112,A -85,B 0,C 180,E1 -2003.11,E2 -2003.11} C_VEL
LIN {X 0,Y 573.017,Z 491.31,A -85,B 0,C 180,E1 -2003.875,E2 -2003.875} C_VEL
LIN {X 0,Y 573.025,Z 486.724,A -85,B 0,C 180,E1 -2004.835,E2 -2004.835} C_VEL
LIN {X 0,Y 573.061,Z 482.018,A -85,B 0,C 180,E1 -2005.614,E2 -2005.614} C_VEL
LIN {X 0,Y 573.094,Z 476.726,A -85,B 0,C 180,E1 -2006.336,E2 -2006.336} C_VEL
LIN {X 0,Y 573.113,Z 471.057,A -85,B 0,C 180,E1 -2006.983,E2 -2006.983} C_VEL
LIN {X 0,Y 573.197,Z 463.806,A -85,B 0,C 180,E1 -2007.671,E2 -2007.671} C_VEL
LIN {X 0,Y 573.277,Z 455.173,A -85,B 0,C 180,E1 -2008.337,E2 -2008.337} C_VEL
LIN {X 0,Y 573.398,Z 443.86,A -85,B 0,C 180,E1 -2009.007,E2 -2009.007} C_VEL
LIN {X 0,Y 573.457,Z 434.84,A -85,B 0,C 180,E1 -2009.408,E2 -2009.408} C_VEL
LIN {X 0,Y 573.469,Z 424.95,A -85,B 0,C 180,E1 -2009.732,E2 -2009.732} C_VEL
LIN {X 0,Y 573.525,Z 415.357,A -85,B 0,C 180,E1 -2009.942,E2 -2009.942} C_VEL
LIN {X 0,Y 573.62,Z 342.235,A -85,B 0,C 180,E1 -2010.869,E2 -2010.869} C_VEL
LIN {X 0,Y 573.189,Z 338.679,A -85,B 0,C 180,E1 -2010.929,E2 -2010.929} C_VEL
LIN {X 0,Y 573.291,Z 320.105,A -85,B 0,C 180,E1 -2013.903,E2 -2013.903} C_VEL
LIN {X 0,Y 573.421,Z 305.568,A -85,B 0,C 180,E1 -2016.254,E2 -2016.254} C_VEL
LIN {X 0,Y 573.576,Z 289.545,A -85,B 0,C 180,E1 -2018.878,E2 -2018.878} C_VEL
LIN {X 0,Y 573.736,Z 272.66,A -85,B 0,C 180,E1 -2021.654,E2 -2021.654} C_VEL
LIN {X 0,Y 573.241,Z 269.081,A -85,B 0,C 180,E1 -2022.294,E2 -2022.294} C_VEL
LIN {X 0,Y 573.202,Z 269.086,A -85,B 0,C 180,E1 -2025.328,E2 -2025.328} C_VEL
LIN {X 0,Y 573.229,Z 269.08,A -85,B 0,C 180,E1 -2027.602,E2 -2027.602} C_VEL
LIN {X 0,Y 573.227,Z 269.074,A -85,B 0,C 180,E1 -2030.571,E2 -2030.571} C_VEL
LIN {X 0,Y 573.217,Z 269.078,A -85,B 0,C 180,E1 -2033.077,E2 -2033.077} C_VEL
LIN {X 0,Y 573.249,Z 269.081,A -85,B 0,C 180,E1 -2035.672,E2 -2035.672} C_VEL
LIN {X 0,Y 573.229,Z 269.08,A -85,B 0,C 180,E1 -2038.186,E2 -2038.186} C_VEL
LIN {X 0,Y 573.219,Z 269.077,A -85,B 0,C 180,E1 -2040.633,E2 -2040.633} C_VEL
LIN {X 0,Y 573.204,Z 269.078,A -85,B 0,C 180,E1 -2043.515,E2 -2043.515} C_VEL
LIN {X 0,Y 573.194,Z 269.085,A -85,B 0,C 180,E1 -2046.134,E2 -2046.134} C_VEL
LIN {X 0,Y 573.227,Z 269.075,A -85,B 0,C 180,E1 -2049.173,E2 -2049.173} C_VEL
LIN {X 0,Y 573.197,Z 269.078,A -85,B 0,C 180,E1 -2051.411,E2 -2051.411} C_VEL
LIN {X 0,Y 573.225,Z 269.074,A -85,B 0,C 180,E1 -2053.621,E2 -2053.621} C_VEL
LIN {X 0,Y 573.203,Z 269.081,A -85,B 0,C 180,E1 -2056.529,E2 -2056.529} C_VEL
LIN {X 0,Y 573.244,Z 269.078,A -85,B 0,C 180,E1 -2059.403,E2 -2059.403} C_VEL
LIN {X 0,Y 573.213,Z 269.076,A -85,B 0,C 180,E1 -2062.248,E2 -2062.248} C_VEL
LIN {X 0,Y 573.293,Z 269.07,A -85,B 0,C 180,E1 -2065.076,E2 -2065.076} C_VEL
LIN {X 0,Y 573.302,Z 269.071,A -85,B 0,C 180,E1 -2067.891,E2 -2067.891} C_VEL
LIN {X 0,Y 573.319,Z 269.069,A -85,B 0,C 180,E1 -2069.999,E2 -2069.999} C_VEL
LIN {X 0,Y 573.271,Z 269.068,A -85,B 0,C 180,E1 -2072.809,E2 -2072.809} C_VEL
LIN {X 0,Y 573.259,Z 269.074,A -85,B 0,C 180,E1 -2075.626,E2 -2075.626} C_VEL
LIN {X 0,Y 573.235,Z 269.08,A -85,B 0,C 180,E1 -2078.458,E2 -2078.458} C_VEL
LIN {X 0,Y 573.271,Z 269.068,A -85,B 0,C 180,E1 -2081.309,E2 -2081.309} C_VEL
LIN {X 0,Y 573.251,Z 269.08,A -85,B 0,C 180,E1 -2084.41,E2 -2084.41} C_VEL
LIN {X 0,Y 573.249,Z 269.076,A -85,B 0,C 180,E1 -2087.109,E2 -2087.109} C_VEL
LIN {X 0,Y 573.222,Z 269.075,A -85,B 0,C 180,E1 -2090.074,E2 -2090.074} C_VEL
LIN {X 0,Y 573.207,Z 269.078,A -85,B 0,C 180,E1 -2092.335,E2 -2092.335} C_VEL
LIN {X 0,Y 573.217,Z 269.082,A -85,B 0,C 180,E1 -2095.408,E2 -2095.408} C_VEL
LIN {X 0,Y 573.203,Z 269.077,A -85,B 0,C 180,E1 -2098.562,E2 -2098.562} C_VEL
LIN {X 0,Y 573.197,Z 269.08,A -85,B 0,C 180,E1 -2100.99,E2 -2100.99} C_VEL
LIN {X 0,Y 573.241,Z 269.081,A -85,B 0,C 180,E1 -2103.52,E2 -2103.52} C_VEL
LIN {X 0,Y 573.215,Z 269.082,A -85,B 0,C 180,E1 -2106.046,E2 -2106.046} C_VEL
LIN {X 0,Y 573.212,Z 269.077,A -85,B 0,C 180,E1 -2108.698,E2 -2108.698} C_VEL
LIN {X 0,Y 573.211,Z 269.079,A -85,B 0,C 180,E1 -2111.59,E2 -2111.59} C_VEL
LIN {X 0,Y 573.193,Z 269.089,A -85,B 0,C 180,E1 -2114.33,E2 -2114.33} C_VEL
LIN {X 0,Y 573.198,Z 269.078,A -85,B 0,C 180,E1 -2117.355,E2 -2117.355} C_VEL
LIN {X 0,Y 573.234,Z 269.073,A -85,B 0,C 180,E1 -2119.473,E2 -2119.473} C_VEL
LIN {X 0,Y 573.191,Z 269.081,A -85,B 0,C 180,E1 -2122.188,E2 -2122.188} C_VEL
LIN {X 0,Y 573.22,Z 269.085,A -85,B 0,C 180,E1 -2124.813,E2 -2124.813} C_VEL
LIN {X 0,Y 573.206,Z 269.077,A -85,B 0,C 180,E1 -2127.767,E2 -2127.767} C_VEL
LIN {X 0,Y 573.228,Z 269.076,A -85,B 0,C 180,E1 -2130.632,E2 -2130.632} C_VEL
LIN {X 0,Y 573.216,Z 269.085,A -85,B 0,C 180,E1 -2133.497,E2 -2133.497} C_VEL
LIN {X 0,Y 573.19,Z 269.08,A -85,B 0,C 180,E1 -2136.132,E2 -2136.132} C_VEL
LIN {X 0,Y 573.202,Z 269.077,A -85,B 0,C 180,E1 -2138.703,E2 -2138.703} C_VEL
LIN {X 0,Y 573.184,Z 269.083,A -85,B 0,C 180,E1 -2141.41,E2 -2141.41} C_VEL
LIN {X 0,Y 573.208,Z 269.082,A -85,B 0,C 180,E1 -2143.62,E2 -2143.62} C_VEL
LIN {X 0,Y 573.235,Z 269.079,A -85,B 0,C 180,E1 -2145.806,E2 -2145.806} C_VEL
LIN {X 0,Y 573.196,Z 269.081,A -85,B 0,C 180,E1 -2148.743,E2 -2148.743} C_VEL
LIN {X 0,Y 573.244,Z 269.072,A -85,B 0,C 180,E1 -2151.54,E2 -2151.54} C_VEL
LIN {X 0,Y 573.261,Z 269.077,A -85,B 0,C 180,E1 -2154.371,E2 -2154.371} C_VEL
LIN {X 0,Y 573.253,Z 269.074,A -85,B 0,C 180,E1 -2157.189,E2 -2157.189} C_VEL
LIN {X 0,Y 573.247,Z 269.072,A -85,B 0,C 180,E1 -2160,E2 -2160} C_VEL
LIN {X 0,Y 573.256,Z 269.077,A -85,B 0,C 180,E1 -2162.81,E2 -2162.81} C_VEL
LIN {X 0,Y 573.258,Z 269.074,A -85,B 0,C 180,E1 -2165.628,E2 -2165.628} C_VEL
LIN {X 0,Y 573.242,Z 269.072,A -85,B 0,C 180,E1 -2168.46,E2 -2168.46} C_VEL
LIN {X 0,Y 573.204,Z 269.084,A -85,B 0,C 180,E1 -2171.313,E2 -2171.313} C_VEL
LIN {X 0,Y 573.233,Z 269.076,A -85,B 0,C 180,E1 -2174.194,E2 -2174.194} C_VEL
LIN {X 0,Y 573.195,Z 269.078,A -85,B 0,C 180,E1 -2177.113,E2 -2177.113} C_VEL
LIN {X 0,Y 573.198,Z 269.089,A -85,B 0,C 180,E1 -2180.078,E2 -2180.078} C_VEL
LIN {X 0,Y 573.211,Z 269.076,A -85,B 0,C 180,E1 -2183.156,E2 -2183.156} C_VEL
LIN {X 0,Y 573.229,Z 269.081,A -85,B 0,C 180,E1 -2186.191,E2 -2186.191} C_VEL
LIN {X 0,Y 573.192,Z 269.09,A -85,B 0,C 180,E1 -2188.567,E2 -2188.567} C_VEL
LIN {X 0,Y 573.17,Z 269.086,A -85,B 0,C 180,E1 -2190.996,E2 -2190.996} C_VEL
LIN {X 0,Y 573.21,Z 269.077,A -85,B 0,C 180,E1 -2193.527,E2 -2193.527} C_VEL
LIN {X 0,Y 573.202,Z 269.077,A -85,B 0,C 180,E1 -2196.052,E2 -2196.052} C_VEL
LIN {X 0,Y 573.197,Z 269.082,A -85,B 0,C 180,E1 -2198.705,E2 -2198.705} C_VEL
LIN {X 0,Y 573.181,Z 269.085,A -85,B 0,C 180,E1 -2201.596,E2 -2201.596} C_VEL
LIN {X 0,Y 573.186,Z 269.079,A -85,B 0,C 180,E1 -2204.338,E2 -2204.338} C_VEL
LIN {X 0,Y 573.206,Z 269.083,A -85,B 0,C 180,E1 -2207.362,E2 -2207.362} C_VEL
LIN {X 0,Y 573.199,Z 269.079,A -85,B 0,C 180,E1 -2210.396,E2 -2210.396} C_VEL
LIN {X 0,Y 573.193,Z 269.078,A -85,B 0,C 180,E1 -2213.079,E2 -2213.079} C_VEL
LIN {X 0,Y 573.225,Z 269.078,A -85,B 0,C 180,E1 -2215.674,E2 -2215.674} C_VEL
LIN {X 0,Y 573.196,Z 269.089,A -85,B 0,C 180,E1 -2218.187,E2 -2218.187} C_VEL
LIN {X 0,Y 573.196,Z 269.085,A -85,B 0,C 180,E1 -2220.635,E2 -2220.635} C_VEL
LIN {X 0,Y 573.18,Z 269.081,A -85,B 0,C 180,E1 -2223.518,E2 -2223.518} C_VEL
LIN {X 0,Y 573.17,Z 269.087,A -85,B 0,C 180,E1 -2226.136,E2 -2226.136} C_VEL
LIN {X 0,Y 573.189,Z 269.153,A -85,B 0,C 180,E1 -2227.004,E2 -2227.004} C_VEL
LIN {X 0,Y 574.205,Z 274.591,A -85,B 0,C 180,E1 -2227.706,E2 -2227.706} C_VEL
LIN {X 0,Y 573.975,Z 297.985,A -85,B 0,C 180,E1 -2230.53,E2 -2230.53} C_VEL
LIN {X 0,Y 573.7,Z 322.541,A -85,B 0,C 180,E1 -2233.455,E2 -2233.455} C_VEL
LIN {X 0,Y 573.483,Z 345.581,A -85,B 0,C 180,E1 -2236.154,E2 -2236.154} C_VEL
LIN {X 0,Y 574.078,Z 350.946,A -85,B 0,C 180,E1 -2236.237,E2 -2236.237} C_VEL
LIN {X 0,Y 573.864,Z 454.752,A -85,B 0,C 180,E1 -2237.56,E2 -2237.56} C_VEL
LIN {X 0,Y 573.774,Z 465.794,A -85,B 0,C 180,E1 -2237.805,E2 -2237.805} C_VEL
LIN {X 0,Y 573.698,Z 476.046,A -85,B 0,C 180,E1 -2238.13,E2 -2238.13} C_VEL
LIN {X 0,Y 573.647,Z 486.17,A -85,B 0,C 180,E1 -2238.553,E2 -2238.553} C_VEL
